(* CODESYS project xlh_gantry_example_1_00_02.project
   Author: 3S - Smart Software Solutions GmbH
   Version: 1.0.0.0
   Description: Receives some incoming messages and echoes them with CAN-ID +1
   Title: CAN Bus API Example
   Company: 3S - Smart Software Solutions GmbH

Project tree, tasks and I/O mapping:
  xLH_base : CODESYS Control for Raspberry Pi 64 SL, CODESYS, order no. 2302000009, version 4.20.0.0
    application app
      libraries: Standard, 3.5.22.0 (System); Util, 3.5.22.0 (System); VisuDialogs, * (System); Memory, * (3S - Smart Software Solutions GmbH); CmpBitmapPool, * (System); MemoryUtils, * (3S - Smart Software Solutions GmbH); CAA CiA 405, 4.3.0.0 (CODESYS)
      task CANOPEN_TASK (cyclic, interval 1 ms, priority 1) calls nothing
      task VISU_TASK (cyclic, interval 100 ms, priority 31) calls VisuElems.Visu_Prg
      task MAIN_TASK (cyclic, interval 4 ms, priority 2) calls io, MAIN_CALLER
      task SoftMotion_PlanningTask (cyclic, interval t#2ms, priority 15) calls nothing
      program MAIN_CALLER [ST]
      visualisation Visualization
      data type MOTION_CONTROL_BYTE
      MOTION_BASE/
        function block FB_XLH_MOTION_AXIS_SIMPLE_ES [ST]: mRead
        function block FB_PLC_OPEN_AXIS [ST]: plcOpen, executeToFalse
        function block FB_XLH_MOTION_AXIS_SIMPLE [ST]
        function block FB_XLH_MOTION_AXIS_BASE [ST]: mRead, mWrite
        function block FB_AXG_MOVE_ABSOLUTE [ST]
        function block FB_AXG_MOVE_RELATIVE [ST]
        function block FB_AXG_PICK_AND_PLACE [ST]: moveToOffset, setMagnet
        function block FB_KALMAN_FILTER [ST]: reset
        data type ST_PnpStep
      IO/
        function block FB_XLH_MOTION [ST]: read, write
        program io [ST]: read, write
        function block FB_XLH_GPIO [ST]: read, write
        function block FB_XLH_TERMINAL [ST]: read, write
        data type RGB
        data type UNION_BYTE_INT
        trace RT (task MAIN_TASK): io.terminal.bRtMagnet, io.terminal.bMagnet, MANUAL_MODE.iDummy
      program MC [ST]: write_io, read_io, axSmExecuteToFalse, axGexecuteToFalse, axInitPointers, axPowerOn, axStartHomingZA, axStopHoming, axCmdReset, axSetDefaultKinValues, axStartHomingXY, homing
      axis group AxisGroup: TRAFO.Kin_Gantry3, axes x_axis, y_axis, z_axis
      GCODE/
        text DEMO_GCODE
      CNC settings
      program MANUAL_MODE [ST]: TODO
      program CNC_MODE [ST]
      program APP_SQUARE_MODE [ST]
      MISC/
        TRACE/
          trace Trace_AxX (task MAIN_TASK): x_axis.fActPosition, x_axis.fSetPosition, x_axis.fSetAcceleration, x_axis.fActAcceleration, x_axis.fSetVelocity, x_axis.fActVelocity, io.motion.adiFrequency[1]
          trace Trace (task MAIN_TASK): MC.diPosition, MC.iSetSpeed, MC.iDebug2Pos, MC.iDebug1Mileage, MC.auiUltrasonic[1], MC.fbReadStatusLoopTime.udiValue, MC.iSpeed2, MC.iSpeed1, MC.iPitch
          trace Trace_AxZ (task MAIN_TASK): z_axis.fActPosition, z_axis.fSetPosition, z_axis.fSetAcceleration, z_axis.fActAcceleration, z_axis.fSetVelocity, z_axis.fActVelocity, io.motion.adiFrequency[3]
    CANbus : CANbus, CODESYS, version 4.3.0.0
        settings: Baudrate = 1000 kbit/s
      CANopen_Manager : CANopen_Manager, CODESYS, version 4.3.0.0
          settings: NMT Start All = TRUE; Polling of optional slaves = FALSE; ConfigVersion = 50659584
        xlh_motion : xlh_motion, xemax ag, order no. 0, version Revision=16#00000001, FileVersion=1.0
            settings: NODEIDSAVED = 1; SDO Timeout = 1000000; PDO_Autoconfig = FALSE; EXPERTSETTINGS = True; Sync-General Parameters.Sync-COBID = 16#00000080; Sync-General Parameters.Communication Cycle Period = 16#00000000 usec; PDO 16#1400.COBID = 16#00000201; Process by CANopenManager = TRUE; PDO 16#1401.COBID = 16#00000301; Process by CANopenManager = TRUE; PDO 16#1402.COBID = 16#00000401; Process by CANopenManager = TRUE; PDO 16#1403.COBID = 16#00000501; Process by CANopenManager = TRUE; PDO 16#1800.COBID = 16#00000181; Process by CANopenManager = TRUE; PDO 16#1801.COBID = 16#00000281; Process by CANopenManager = TRUE; PDO 16#1802.COBID = 16#00000381; Process by CANopenManager = TRUE; Control 1.Subindex = 16#01; Control 2.Subindex = 16#02; Control 3.Subindex = 16#03; Control 4.Subindex = 16#04; Outputs 0-7.Subindex = 16#01; Outputs 8-15.Subindex = 16#02; Magnet Duty Cycle.Subindex = 16#01; Freqeuncy 1.Subindex = 16#05; Freqeuncy 2.Subindex = 16#06; Freqeuncy 3.Subindex = 16#07; Freqeuncy 4.Subindex = 16#08; Servo 1.Subindex = 16#01; Servo 2.Subindex = 16#02; Servo 3.Subindex = 16#03; Servo 4.Subindex = 16#04; Servo 5.Subindex = 16#05; Servo 6.Subindex = 16#06; Servo 7.Subindex = 16#07; Servo 8.Subindex = 16#08; Position 1.Subindex = 16#01;
              Position 2.Subindex = 16#02; Position 3.Subindex = 16#03; Position 4.Subindex = 16#04; Inputs 0-7.Subindex = 16#01; Inputs 8-15.Subindex = 16#02; Inputs CLK.Subindex = 16#03; SDO List.Set COB-ID sync.Index = 16#1005; SDO List.Set COB-ID sync.Subindex = 16#00; SDO List.Set COB-ID sync.Value = 16#00000080; SDO List.Set COB-ID sync.Size = 32; SDO List.Set COB-ID sync.AbortIfError = FALSE; SDO List.Set COB-ID sync.JumpToLine = FALSE; SDO List.Set COB-ID sync.Line = 0; SDO List.Set communication cycle period.Index = 16#1006; SDO List.Set communication cycle period.Subindex = 16#00; SDO List.Set communication cycle period.Value = 16#00000000; SDO List.Set communication cycle period.Size = 32; SDO List.Set communication cycle period.AbortIfError = FALSE; SDO List.Set communication cycle period.JumpToLine = FALSE; SDO List.Set communication cycle period.Line = 0; SDO List.Set Guardtime.Index = 16#100C; SDO List.Set Guardtime.Subindex = 16#00; SDO List.Set Guardtime.Value = 16#000000C8; SDO List.Set Guardtime.Size = 16; SDO List.Set Guardtime.AbortIfError = FALSE; SDO List.Set Guardtime.JumpToLine = FALSE; SDO List.Set Guardtime.Line = 0; SDO List.Set Lifetime.Index = 16#100D; SDO List.Set Lifetime.Subindex = 16#00; SDO List.Set Lifetime.Value = 16#00000003; SDO List.Set Lifetime.Size = 8; SDO List.Set Lifetime.AbortIfError = FALSE; SDO List.Set Lifetime.JumpToLine = FALSE; SDO List.Set Lifetime.Line = 0; SDO List.Set Heartbeat Consumer.Index = 16#1016; SDO List.Set Heartbeat Consumer.Subindex = 16#01; SDO List.Set Heartbeat Consumer.Value = 0; SDO List.Set Heartbeat Consumer.Size = 32; SDO List.Set Heartbeat Consumer.AbortIfError = FALSE; SDO List.Set Heartbeat Consumer.JumpToLine = FALSE;
              SDO List.Set Heartbeat Consumer.Line = 0; SDO List.Disable PDO.Index = 16#1400; SDO List.Disable PDO.Subindex = 16#01; SDO List.Disable PDO.Value = 16#80000201; SDO List.Disable PDO.Size = 32; SDO List.Disable PDO.AbortIfError = FALSE; SDO List.Disable PDO.JumpToLine = FALSE; SDO List.Disable PDO.Line = 0; SDO List.Set transmission type.Index = 16#1400; SDO List.Set transmission type.Subindex = 16#02; SDO List.Set transmission type.Value = 16#FF; SDO List.Set transmission type.Size = 8; SDO List.Set transmission type.AbortIfError = FALSE; SDO List.Set transmission type.JumpToLine = FALSE; SDO List.Set transmission type.Line = 0; SDO List.Set and enable COB-ID.Index = 16#1400; SDO List.Set and enable COB-ID.Subindex = 16#01; SDO List.Set and enable COB-ID.Value = 16#00000201; SDO List.Set and enable COB-ID.Size = 32; SDO List.Set and enable COB-ID.AbortIfError = FALSE; SDO List.Set and enable COB-ID.JumpToLine = FALSE; SDO List.Set and enable COB-ID.Line = 0; SDO List.Disable PDO.Index = 16#1401; SDO List.Disable PDO.Subindex = 16#01; SDO List.Disable PDO.Value = 16#80000301; SDO List.Disable PDO.Size = 32; SDO List.Disable PDO.AbortIfError = FALSE; SDO List.Disable PDO.JumpToLine = FALSE; SDO List.Disable PDO.Line = 0; SDO List.Set transmission type.Index = 16#1401; SDO List.Set transmission type.Subindex = 16#02; SDO List.Set transmission type.Value = 16#FF; SDO List.Set transmission type.Size = 8; SDO List.Set transmission type.AbortIfError = FALSE; SDO List.Set transmission type.JumpToLine = FALSE; SDO List.Set transmission type.Line = 0; SDO List.Set and enable COB-ID.Index = 16#1401; SDO List.Set and enable COB-ID.Subindex = 16#01; SDO List.Set and enable COB-ID.Value = 16#00000301; SDO List.Set and enable COB-ID.Size = 32;
              SDO List.Set and enable COB-ID.AbortIfError = FALSE; SDO List.Set and enable COB-ID.JumpToLine = FALSE; SDO List.Set and enable COB-ID.Line = 0; SDO List.Disable PDO.Index = 16#1402; SDO List.Disable PDO.Subindex = 16#01; SDO List.Disable PDO.Value = 16#80000401; SDO List.Disable PDO.Size = 32; SDO List.Disable PDO.AbortIfError = FALSE; SDO List.Disable PDO.JumpToLine = FALSE; SDO List.Disable PDO.Line = 0; SDO List.Set transmission type.Index = 16#1402; SDO List.Set transmission type.Subindex = 16#02; SDO List.Set transmission type.Value = 16#FF; SDO List.Set transmission type.Size = 8; SDO List.Set transmission type.AbortIfError = FALSE; SDO List.Set transmission type.JumpToLine = FALSE; SDO List.Set transmission type.Line = 0; SDO List.Set and enable COB-ID.Index = 16#1402; SDO List.Set and enable COB-ID.Subindex = 16#01; SDO List.Set and enable COB-ID.Value = 16#00000401; SDO List.Set and enable COB-ID.Size = 32; SDO List.Set and enable COB-ID.AbortIfError = FALSE; SDO List.Set and enable COB-ID.JumpToLine = FALSE; SDO List.Set and enable COB-ID.Line = 0; SDO List.Disable PDO.Index = 16#1403; SDO List.Disable PDO.Subindex = 16#01; SDO List.Disable PDO.Value = 16#80000501; SDO List.Disable PDO.Size = 32; SDO List.Disable PDO.AbortIfError = FALSE; SDO List.Disable PDO.JumpToLine = FALSE; SDO List.Disable PDO.Line = 0; SDO List.Set transmission type.Index = 16#1403; SDO List.Set transmission type.Subindex = 16#02; SDO List.Set transmission type.Value = 16#FF; SDO List.Set transmission type.Size = 8; SDO List.Set transmission type.AbortIfError = FALSE; SDO List.Set transmission type.JumpToLine = FALSE; SDO List.Set transmission type.Line = 0; SDO List.Set and enable COB-ID.Index = 16#1403; SDO List.Set and enable COB-ID.Subindex = 16#01;
              SDO List.Set and enable COB-ID.Value = 16#00000501; SDO List.Set and enable COB-ID.Size = 32; SDO List.Set and enable COB-ID.AbortIfError = FALSE; SDO List.Set and enable COB-ID.JumpToLine = FALSE; SDO List.Set and enable COB-ID.Line = 0; SDO List.Disable PDO.Index = 16#1800; SDO List.Disable PDO.Subindex = 16#01; SDO List.Disable PDO.Value = 16#80000181; SDO List.Disable PDO.Size = 32; SDO List.Disable PDO.AbortIfError = FALSE; SDO List.Disable PDO.JumpToLine = FALSE; SDO List.Disable PDO.Line = 0; SDO List.Set transmission type.Index = 16#1800; SDO List.Set transmission type.Subindex = 16#02; SDO List.Set transmission type.Value = 16#FF; SDO List.Set transmission type.Size = 8; SDO List.Set transmission type.AbortIfError = FALSE; SDO List.Set transmission type.JumpToLine = FALSE; SDO List.Set transmission type.Line = 0; SDO List.Set inhibit time.Index = 16#1800; SDO List.Set inhibit time.Subindex = 16#03; SDO List.Set inhibit time.Value = 16#0000; SDO List.Set inhibit time.Size = 16; SDO List.Set inhibit time.AbortIfError = FALSE; SDO List.Set inhibit time.JumpToLine = FALSE; SDO List.Set inhibit time.Line = 0; SDO List.Set event time.Index = 16#1800; SDO List.Set event time.Subindex = 16#05; SDO List.Set event time.Value = 16#0000; SDO List.Set event time.Size = 16; SDO List.Set event time.AbortIfError = FALSE; SDO List.Set event time.JumpToLine = FALSE; SDO List.Set event time.Line = 0; SDO List.Set and enable COB-ID.Index = 16#1800; SDO List.Set and enable COB-ID.Subindex = 16#01; SDO List.Set and enable COB-ID.Value = 16#00000181; SDO List.Set and enable COB-ID.Size = 32; SDO List.Set and enable COB-ID.AbortIfError = FALSE; SDO List.Set and enable COB-ID.JumpToLine = FALSE; SDO List.Set and enable COB-ID.Line = 0;
              SDO List.Disable PDO.Index = 16#1801; SDO List.Disable PDO.Subindex = 16#01; SDO List.Disable PDO.Value = 16#80000281; SDO List.Disable PDO.Size = 32; SDO List.Disable PDO.AbortIfError = FALSE; SDO List.Disable PDO.JumpToLine = FALSE; SDO List.Disable PDO.Line = 0; SDO List.Set transmission type.Index = 16#1801; SDO List.Set transmission type.Subindex = 16#02; SDO List.Set transmission type.Value = 16#FF; SDO List.Set transmission type.Size = 8; SDO List.Set transmission type.AbortIfError = FALSE; SDO List.Set transmission type.JumpToLine = FALSE; SDO List.Set transmission type.Line = 0; SDO List.Set inhibit time.Index = 16#1801; SDO List.Set inhibit time.Subindex = 16#03; SDO List.Set inhibit time.Value = 16#0000; SDO List.Set inhibit time.Size = 16; SDO List.Set inhibit time.AbortIfError = FALSE; SDO List.Set inhibit time.JumpToLine = FALSE; SDO List.Set inhibit time.Line = 0; SDO List.Set event time.Index = 16#1801; SDO List.Set event time.Subindex = 16#05; SDO List.Set event time.Value = 16#0000; SDO List.Set event time.Size = 16; SDO List.Set event time.AbortIfError = FALSE; SDO List.Set event time.JumpToLine = FALSE; SDO List.Set event time.Line = 0; SDO List.Set and enable COB-ID.Index = 16#1801; SDO List.Set and enable COB-ID.Subindex = 16#01; SDO List.Set and enable COB-ID.Value = 16#00000281; SDO List.Set and enable COB-ID.Size = 32; SDO List.Set and enable COB-ID.AbortIfError = FALSE; SDO List.Set and enable COB-ID.JumpToLine = FALSE; SDO List.Set and enable COB-ID.Line = 0; SDO List.Disable PDO.Index = 16#1802; SDO List.Disable PDO.Subindex = 16#01; SDO List.Disable PDO.Value = 16#80000381; SDO List.Disable PDO.Size = 32; SDO List.Disable PDO.AbortIfError = FALSE;
              SDO List.Disable PDO.JumpToLine = FALSE; SDO List.Disable PDO.Line = 0; SDO List.Set transmission type.Index = 16#1802; SDO List.Set transmission type.Subindex = 16#02; SDO List.Set transmission type.Value = 16#FF; SDO List.Set transmission type.Size = 8; SDO List.Set transmission type.AbortIfError = FALSE; SDO List.Set transmission type.JumpToLine = FALSE; SDO List.Set transmission type.Line = 0; SDO List.Set inhibit time.Index = 16#1802; SDO List.Set inhibit time.Subindex = 16#03; SDO List.Set inhibit time.Value = 16#0000; SDO List.Set inhibit time.Size = 16; SDO List.Set inhibit time.AbortIfError = FALSE; SDO List.Set inhibit time.JumpToLine = FALSE; SDO List.Set inhibit time.Line = 0; SDO List.Set event time.Index = 16#1802; SDO List.Set event time.Subindex = 16#05; SDO List.Set event time.Value = 16#0000; SDO List.Set event time.Size = 16; SDO List.Set event time.AbortIfError = FALSE; SDO List.Set event time.JumpToLine = FALSE; SDO List.Set event time.Line = 0; SDO List.Set and enable COB-ID.Index = 16#1802; SDO List.Set and enable COB-ID.Subindex = 16#01; SDO List.Set and enable COB-ID.Value = 16#00000381; SDO List.Set and enable COB-ID.Size = 32; SDO List.Set and enable COB-ID.AbortIfError = FALSE; SDO List.Set and enable COB-ID.JumpToLine = FALSE; SDO List.Set and enable COB-ID.Line = 0; ConfigVersion = 50659584
            output app.io.motion.abyControl[1] : USINT  // Control 1
            output app.io.motion.abyControl[2] : USINT  // Control 2
            output app.io.motion.abyControl[3] : USINT  // Control 3
            output app.io.motion.abyControl[4] : USINT  // Control 4
            output app.io.motion.abyOutputs[1] : USINT  // Outputs 0-7
            output app.io.motion.abyOutputs[2] : USINT  // Outputs 8-15
            output app.io.motion.uiMagnetDutyCycle : UINT  // Magnet Duty Cycle
            output app.io.motion.adiFrequency[1] : DINT  // Freqeuncy 1
            output app.io.motion.adiFrequency[2] : DINT  // Freqeuncy 2
            output app.io.motion.adiFrequency[3] : DINT  // Freqeuncy 3
            output app.io.motion.adiFrequency[4] : DINT  // Freqeuncy 4
            output app.io.motion.ausServo[1] : USINT  // Servo 1
            output app.io.motion.ausServo[2] : USINT  // Servo 2
            output app.io.motion.ausServo[3] : USINT  // Servo 3
            output app.io.motion.ausServo[4] : USINT  // Servo 4
            output app.io.motion.ausServo[5] : USINT  // Servo 5
            output app.io.motion.ausServo[6] : USINT  // Servo 6
            output app.io.motion.ausServo[7] : USINT  // Servo 7
            output app.io.motion.ausServo[8] : USINT  // Servo 8
            input  app.io.motion.adiPosition[1] : DINT  // Position 1
            input  app.io.motion.adiPosition[2] : DINT  // Position 2
            input  app.io.motion.adiPosition[3] : DINT  // Position 3
            input  app.io.motion.adiPosition[4] : DINT  // Position 4
            input  app.io.motion.abyInputs[1] : USINT  // Inputs 0-7
            input  app.io.motion.bAxXsw : BOOL  // Inputs 0-7.Bit0
            input  app.io.motion.bAxYsw : BOOL  // Inputs 0-7.Bit1
            input  app.io.motion.bAxZsw : BOOL  // Inputs 0-7.Bit2
            input  app.io.motion._bSensorHw : BOOL  // Inputs 0-7.Bit3
            input  app.io.motion._bSensorConveyorFrontHw : BOOL  // Inputs 0-7.Bit4
            input  app.io.motion._bSensorConveyorBackHw : BOOL  // Inputs 0-7.Bit5
            input  app.io.motion.abyInputs[2] : USINT  // Inputs 8-15
            input  app.io.motion.abyInputs[3] : USINT  // Inputs CLK
        xlh_terminal : xlh_terminal, xemax ag, order no. 0, version Revision=16#00000001, FileVersion=1.0
            settings: NODEIDSAVED = 2; SDO Timeout = 1000000; PDO_Autoconfig = FALSE; EXPERTSETTINGS = FALSE; Nodeguarding.Guard Time = 1000 ms; PDO 16#1400.COBID = 16#00000202; Process by CANopenManager = TRUE; PDO 16#1401.COBID = 16#00000302; Process by CANopenManager = TRUE; PDO 16#1402.COBID = 16#00000402; Process by CANopenManager = TRUE; PDO 16#1403.COBID = 16#00000502; Process by CANopenManager = TRUE; PDO 16#1800.COBID = 16#00000182; Process by CANopenManager = TRUE; PDO 16#1801.COBID = 16#00000282; Process by CANopenManager = TRUE; PDO 16#1802.COBID = 16#00000382; Process by CANopenManager = TRUE; PDO 16#1803.COBID = 16#00000482; Process by CANopenManager = TRUE; Data out 1 Byte 0.Subindex = 16#01; Data out 1 Byte 1.Subindex = 16#02; Data out 1 Byte 2.Subindex = 16#03; Data out 1 Byte 3.Subindex = 16#04; Data out 1 Byte 4.Subindex = 16#05; Data out 1 Byte 5.Subindex = 16#06; Data out 1 Byte 6.Subindex = 16#07; Data out 1 Byte 7.Subindex = 16#08; Data out 2 Byte 0.Subindex = 16#01; Data out 2 Byte 1.Subindex = 16#02; Data out 2 Byte 2.Subindex = 16#03; Data out 2 Byte 3.Subindex = 16#04; Data out 2 Byte 4.Subindex = 16#05; Data out 2 Byte 5.Subindex = 16#06; Data out 2 Byte 6.Subindex = 16#07; Data out 2 Byte 7.Subindex = 16#08; Data out 3 Byte 0.Subindex = 16#01; Data out 3 Byte 1.Subindex = 16#02; Data out 3 Byte 2.Subindex = 16#03;
              Data out 3 Byte 3.Subindex = 16#04; Data out 3 Byte 4.Subindex = 16#05; Data out 3 Byte 5.Subindex = 16#06; Data out 3 Byte 6.Subindex = 16#07; Data out 3 Byte 7.Subindex = 16#08; Data out 4 Byte 0.Subindex = 16#01; Data out 4 Byte 1.Subindex = 16#02; Data out 4 Byte 2.Subindex = 16#03; Data out 4 Byte 3.Subindex = 16#04; Data out 4 Byte 4.Subindex = 16#05; Data out 4 Byte 5.Subindex = 16#06; Data out 4 Byte 6.Subindex = 16#07; Data out 4 Byte 7.Subindex = 16#08; Data in 1 Byte 0.Subindex = 16#01; Data in 1 Byte 1.Subindex = 16#02; Data in 1 Byte 2.Subindex = 16#03; Data in 1 Byte 3.Subindex = 16#04; Data in 1 Byte 4.Subindex = 16#05; Data in 1 Byte 5.Subindex = 16#06; Data in 1 Byte 6.Subindex = 16#07; Data in 1 Byte 7.Subindex = 16#08; Data in 2 Byte 0.Subindex = 16#01; Data in 2 Byte 1.Subindex = 16#02; Data in 2 Byte 2.Subindex = 16#03; Data in 2 Byte 3.Subindex = 16#04; Data in 2 Byte 4.Subindex = 16#05; Data in 2 Byte 5.Subindex = 16#06; Data in 2 Byte 6.Subindex = 16#07; Data in 2 Byte 7.Subindex = 16#08; Data in 3 Byte 0.Subindex = 16#01; Data in 3 Byte 1.Subindex = 16#02; Data in 3 Byte 2.Subindex = 16#03; Data in 3 Byte 3.Subindex = 16#04; Data in 3 Byte 4.Subindex = 16#05; Data in 3 Byte 5.Subindex = 16#06; Data in 3 Byte 6.Subindex = 16#07; Data in 3 Byte 7.Subindex = 16#08; Data in 4 Byte 0.Subindex = 16#01; Data in 4 Byte 1.Subindex = 16#02; Data in 4 Byte 2.Subindex = 16#03;
              Data in 4 Byte 3.Subindex = 16#04; Data in 4 Byte 4.Subindex = 16#05; Data in 4 Byte 5.Subindex = 16#06; Data in 4 Byte 6.Subindex = 16#07; Data in 4 Byte 7.Subindex = 16#08; SDO List.Set COB-ID sync.Index = 16#1005; SDO List.Set COB-ID sync.Subindex = 16#00; SDO List.Set COB-ID sync.Value = 16#00000080; SDO List.Set COB-ID sync.Size = 32; SDO List.Set COB-ID sync.AbortIfError = FALSE; SDO List.Set COB-ID sync.JumpToLine = FALSE; SDO List.Set COB-ID sync.Line = 0; SDO List.Set communication cycle period.Index = 16#1006; SDO List.Set communication cycle period.Subindex = 16#00; SDO List.Set communication cycle period.Value = 16#00000000; SDO List.Set communication cycle period.Size = 32; SDO List.Set communication cycle period.AbortIfError = FALSE; SDO List.Set communication cycle period.JumpToLine = FALSE; SDO List.Set communication cycle period.Line = 0; SDO List.Set Guardtime.Index = 16#100C; SDO List.Set Guardtime.Subindex = 16#00; SDO List.Set Guardtime.Value = 16#000003E8; SDO List.Set Guardtime.Size = 16; SDO List.Set Guardtime.AbortIfError = FALSE; SDO List.Set Guardtime.JumpToLine = FALSE; SDO List.Set Guardtime.Line = 0; SDO List.Set Lifetime.Index = 16#100D; SDO List.Set Lifetime.Subindex = 16#00; SDO List.Set Lifetime.Value = 16#00000003; SDO List.Set Lifetime.Size = 8; SDO List.Set Lifetime.AbortIfError = FALSE; SDO List.Set Lifetime.JumpToLine = FALSE; SDO List.Set Lifetime.Line = 0; SDO List.Set Heartbeat Consumer.Index = 16#1016; SDO List.Set Heartbeat Consumer.Subindex = 16#01; SDO List.Set Heartbeat Consumer.Value = 0; SDO List.Set Heartbeat Consumer.Size = 32; SDO List.Set Heartbeat Consumer.AbortIfError = FALSE; SDO List.Set Heartbeat Consumer.JumpToLine = FALSE; SDO List.Set Heartbeat Consumer.Line = 0;
              SDO List.Disable PDO.Index = 16#1400; SDO List.Disable PDO.Subindex = 16#01; SDO List.Disable PDO.Value = 16#80000202; SDO List.Disable PDO.Size = 32; SDO List.Disable PDO.AbortIfError = FALSE; SDO List.Disable PDO.JumpToLine = FALSE; SDO List.Disable PDO.Line = 0; SDO List.Set transmission type.Index = 16#1400; SDO List.Set transmission type.Subindex = 16#02; SDO List.Set transmission type.Value = 16#FF; SDO List.Set transmission type.Size = 8; SDO List.Set transmission type.AbortIfError = FALSE; SDO List.Set transmission type.JumpToLine = FALSE; SDO List.Set transmission type.Line = 0; SDO List.Set and enable COB-ID.Index = 16#1400; SDO List.Set and enable COB-ID.Subindex = 16#01; SDO List.Set and enable COB-ID.Value = 16#00000202; SDO List.Set and enable COB-ID.Size = 32; SDO List.Set and enable COB-ID.AbortIfError = FALSE; SDO List.Set and enable COB-ID.JumpToLine = FALSE; SDO List.Set and enable COB-ID.Line = 0; SDO List.Disable PDO.Index = 16#1401; SDO List.Disable PDO.Subindex = 16#01; SDO List.Disable PDO.Value = 16#80000302; SDO List.Disable PDO.Size = 32; SDO List.Disable PDO.AbortIfError = FALSE; SDO List.Disable PDO.JumpToLine = FALSE; SDO List.Disable PDO.Line = 0; SDO List.Set transmission type.Index = 16#1401; SDO List.Set transmission type.Subindex = 16#02; SDO List.Set transmission type.Value = 16#FF; SDO List.Set transmission type.Size = 8; SDO List.Set transmission type.AbortIfError = FALSE; SDO List.Set transmission type.JumpToLine = FALSE; SDO List.Set transmission type.Line = 0; SDO List.Set and enable COB-ID.Index = 16#1401; SDO List.Set and enable COB-ID.Subindex = 16#01; SDO List.Set and enable COB-ID.Value = 16#00000302; SDO List.Set and enable COB-ID.Size = 32; SDO List.Set and enable COB-ID.AbortIfError = FALSE;
              SDO List.Set and enable COB-ID.JumpToLine = FALSE; SDO List.Set and enable COB-ID.Line = 0; SDO List.Disable PDO.Index = 16#1402; SDO List.Disable PDO.Subindex = 16#01; SDO List.Disable PDO.Value = 16#80000402; SDO List.Disable PDO.Size = 32; SDO List.Disable PDO.AbortIfError = FALSE; SDO List.Disable PDO.JumpToLine = FALSE; SDO List.Disable PDO.Line = 0; SDO List.Set transmission type.Index = 16#1402; SDO List.Set transmission type.Subindex = 16#02; SDO List.Set transmission type.Value = 16#FF; SDO List.Set transmission type.Size = 8; SDO List.Set transmission type.AbortIfError = FALSE; SDO List.Set transmission type.JumpToLine = FALSE; SDO List.Set transmission type.Line = 0; SDO List.Set and enable COB-ID.Index = 16#1402; SDO List.Set and enable COB-ID.Subindex = 16#01; SDO List.Set and enable COB-ID.Value = 16#00000402; SDO List.Set and enable COB-ID.Size = 32; SDO List.Set and enable COB-ID.AbortIfError = FALSE; SDO List.Set and enable COB-ID.JumpToLine = FALSE; SDO List.Set and enable COB-ID.Line = 0; SDO List.Disable PDO.Index = 16#1403; SDO List.Disable PDO.Subindex = 16#01; SDO List.Disable PDO.Value = 16#80000502; SDO List.Disable PDO.Size = 32; SDO List.Disable PDO.AbortIfError = FALSE; SDO List.Disable PDO.JumpToLine = FALSE; SDO List.Disable PDO.Line = 0; SDO List.Set transmission type.Index = 16#1403; SDO List.Set transmission type.Subindex = 16#02; SDO List.Set transmission type.Value = 16#FF; SDO List.Set transmission type.Size = 8; SDO List.Set transmission type.AbortIfError = FALSE; SDO List.Set transmission type.JumpToLine = FALSE; SDO List.Set transmission type.Line = 0; SDO List.Set and enable COB-ID.Index = 16#1403; SDO List.Set and enable COB-ID.Subindex = 16#01; SDO List.Set and enable COB-ID.Value = 16#00000502;
              SDO List.Set and enable COB-ID.Size = 32; SDO List.Set and enable COB-ID.AbortIfError = FALSE; SDO List.Set and enable COB-ID.JumpToLine = FALSE; SDO List.Set and enable COB-ID.Line = 0; SDO List.Disable PDO.Index = 16#1800; SDO List.Disable PDO.Subindex = 16#01; SDO List.Disable PDO.Value = 16#80000182; SDO List.Disable PDO.Size = 32; SDO List.Disable PDO.AbortIfError = FALSE; SDO List.Disable PDO.JumpToLine = FALSE; SDO List.Disable PDO.Line = 0; SDO List.Set transmission type.Index = 16#1800; SDO List.Set transmission type.Subindex = 16#02; SDO List.Set transmission type.Value = 16#FF; SDO List.Set transmission type.Size = 8; SDO List.Set transmission type.AbortIfError = FALSE; SDO List.Set transmission type.JumpToLine = FALSE; SDO List.Set transmission type.Line = 0; SDO List.Set inhibit time.Index = 16#1800; SDO List.Set inhibit time.Subindex = 16#03; SDO List.Set inhibit time.Value = 16#0000; SDO List.Set inhibit time.Size = 16; SDO List.Set inhibit time.AbortIfError = FALSE; SDO List.Set inhibit time.JumpToLine = FALSE; SDO List.Set inhibit time.Line = 0; SDO List.Set event time.Index = 16#1800; SDO List.Set event time.Subindex = 16#05; SDO List.Set event time.Value = 16#0000; SDO List.Set event time.Size = 16; SDO List.Set event time.AbortIfError = FALSE; SDO List.Set event time.JumpToLine = FALSE; SDO List.Set event time.Line = 0; SDO List.Set and enable COB-ID.Index = 16#1800; SDO List.Set and enable COB-ID.Subindex = 16#01; SDO List.Set and enable COB-ID.Value = 16#00000182; SDO List.Set and enable COB-ID.Size = 32; SDO List.Set and enable COB-ID.AbortIfError = FALSE; SDO List.Set and enable COB-ID.JumpToLine = FALSE; SDO List.Set and enable COB-ID.Line = 0; SDO List.Disable PDO.Index = 16#1801;
              SDO List.Disable PDO.Subindex = 16#01; SDO List.Disable PDO.Value = 16#80000282; SDO List.Disable PDO.Size = 32; SDO List.Disable PDO.AbortIfError = FALSE; SDO List.Disable PDO.JumpToLine = FALSE; SDO List.Disable PDO.Line = 0; SDO List.Set transmission type.Index = 16#1801; SDO List.Set transmission type.Subindex = 16#02; SDO List.Set transmission type.Value = 16#FF; SDO List.Set transmission type.Size = 8; SDO List.Set transmission type.AbortIfError = FALSE; SDO List.Set transmission type.JumpToLine = FALSE; SDO List.Set transmission type.Line = 0; SDO List.Set inhibit time.Index = 16#1801; SDO List.Set inhibit time.Subindex = 16#03; SDO List.Set inhibit time.Value = 16#0000; SDO List.Set inhibit time.Size = 16; SDO List.Set inhibit time.AbortIfError = FALSE; SDO List.Set inhibit time.JumpToLine = FALSE; SDO List.Set inhibit time.Line = 0; SDO List.Set event time.Index = 16#1801; SDO List.Set event time.Subindex = 16#05; SDO List.Set event time.Value = 16#0000; SDO List.Set event time.Size = 16; SDO List.Set event time.AbortIfError = FALSE; SDO List.Set event time.JumpToLine = FALSE; SDO List.Set event time.Line = 0; SDO List.Set and enable COB-ID.Index = 16#1801; SDO List.Set and enable COB-ID.Subindex = 16#01; SDO List.Set and enable COB-ID.Value = 16#00000282; SDO List.Set and enable COB-ID.Size = 32; SDO List.Set and enable COB-ID.AbortIfError = FALSE; SDO List.Set and enable COB-ID.JumpToLine = FALSE; SDO List.Set and enable COB-ID.Line = 0; SDO List.Disable PDO.Index = 16#1802; SDO List.Disable PDO.Subindex = 16#01; SDO List.Disable PDO.Value = 16#80000382; SDO List.Disable PDO.Size = 32; SDO List.Disable PDO.AbortIfError = FALSE; SDO List.Disable PDO.JumpToLine = FALSE;
              SDO List.Disable PDO.Line = 0; SDO List.Set transmission type.Index = 16#1802; SDO List.Set transmission type.Subindex = 16#02; SDO List.Set transmission type.Value = 16#FF; SDO List.Set transmission type.Size = 8; SDO List.Set transmission type.AbortIfError = FALSE; SDO List.Set transmission type.JumpToLine = FALSE; SDO List.Set transmission type.Line = 0; SDO List.Set inhibit time.Index = 16#1802; SDO List.Set inhibit time.Subindex = 16#03; SDO List.Set inhibit time.Value = 16#0000; SDO List.Set inhibit time.Size = 16; SDO List.Set inhibit time.AbortIfError = FALSE; SDO List.Set inhibit time.JumpToLine = FALSE; SDO List.Set inhibit time.Line = 0; SDO List.Set event time.Index = 16#1802; SDO List.Set event time.Subindex = 16#05; SDO List.Set event time.Value = 16#0000; SDO List.Set event time.Size = 16; SDO List.Set event time.AbortIfError = FALSE; SDO List.Set event time.JumpToLine = FALSE; SDO List.Set event time.Line = 0; SDO List.Set and enable COB-ID.Index = 16#1802; SDO List.Set and enable COB-ID.Subindex = 16#01; SDO List.Set and enable COB-ID.Value = 16#00000382; SDO List.Set and enable COB-ID.Size = 32; SDO List.Set and enable COB-ID.AbortIfError = FALSE; SDO List.Set and enable COB-ID.JumpToLine = FALSE; SDO List.Set and enable COB-ID.Line = 0; SDO List.Disable PDO.Index = 16#1803; SDO List.Disable PDO.Subindex = 16#01; SDO List.Disable PDO.Value = 16#80000482; SDO List.Disable PDO.Size = 32; SDO List.Disable PDO.AbortIfError = FALSE; SDO List.Disable PDO.JumpToLine = FALSE; SDO List.Disable PDO.Line = 0; SDO List.Set transmission type.Index = 16#1803; SDO List.Set transmission type.Subindex = 16#02; SDO List.Set transmission type.Value = 16#FF; SDO List.Set transmission type.Size = 8;
              SDO List.Set transmission type.AbortIfError = FALSE; SDO List.Set transmission type.JumpToLine = FALSE; SDO List.Set transmission type.Line = 0; SDO List.Set inhibit time.Index = 16#1803; SDO List.Set inhibit time.Subindex = 16#03; SDO List.Set inhibit time.Value = 16#0000; SDO List.Set inhibit time.Size = 16; SDO List.Set inhibit time.AbortIfError = FALSE; SDO List.Set inhibit time.JumpToLine = FALSE; SDO List.Set inhibit time.Line = 0; SDO List.Set event time.Index = 16#1803; SDO List.Set event time.Subindex = 16#05; SDO List.Set event time.Value = 16#0000; SDO List.Set event time.Size = 16; SDO List.Set event time.AbortIfError = FALSE; SDO List.Set event time.JumpToLine = FALSE; SDO List.Set event time.Line = 0; SDO List.Set and enable COB-ID.Index = 16#1803; SDO List.Set and enable COB-ID.Subindex = 16#01; SDO List.Set and enable COB-ID.Value = 16#00000482; SDO List.Set and enable COB-ID.Size = 32; SDO List.Set and enable COB-ID.AbortIfError = FALSE; SDO List.Set and enable COB-ID.JumpToLine = FALSE; SDO List.Set and enable COB-ID.Line = 0; ConfigVersion = 50659584
            output app.io.terminal.abyOutData1[0] : USINT  // Data out 1 Byte 0
            output app.io.terminal.abyOutData1[1] : USINT  // Data out 1 Byte 1
            output app.io.terminal.abyOutData1[2] : USINT  // Data out 1 Byte 2
            output app.io.terminal.abyOutData1[3] : USINT  // Data out 1 Byte 3
            output app.io.terminal.abyOutData1[4] : USINT  // Data out 1 Byte 4
            output app.io.terminal.abyOutData1[5] : USINT  // Data out 1 Byte 5
            output app.io.terminal.abyOutData1[6] : USINT  // Data out 1 Byte 6
            output app.io.terminal.abyOutData1[7] : USINT  // Data out 1 Byte 7
            output app.io.terminal.abyOutData2[0] : USINT  // Data out 2 Byte 0
            output app.io.terminal.abyOutData2[1] : USINT  // Data out 2 Byte 1
            output app.io.terminal.abyOutData2[2] : USINT  // Data out 2 Byte 2
            output app.io.terminal.abyOutData2[3] : USINT  // Data out 2 Byte 3
            output app.io.terminal.abyOutData2[4] : USINT  // Data out 2 Byte 4
            output app.io.terminal.abyOutData2[5] : USINT  // Data out 2 Byte 5
            output app.io.terminal.abyOutData2[6] : USINT  // Data out 2 Byte 6
            output app.io.terminal.abyOutData2[7] : USINT  // Data out 2 Byte 7
            output app.io.terminal.abyOutData3[0] : USINT  // Data out 3 Byte 0
            output app.io.terminal.abyOutData3[1] : USINT  // Data out 3 Byte 1
            output app.io.terminal.abyOutData3[2] : USINT  // Data out 3 Byte 2
            output app.io.terminal.abyOutData3[3] : USINT  // Data out 3 Byte 3
            output app.io.terminal.abyOutData3[4] : USINT  // Data out 3 Byte 4
            output app.io.terminal.abyOutData3[5] : USINT  // Data out 3 Byte 5
            output app.io.terminal.abyOutData3[6] : USINT  // Data out 3 Byte 6
            output app.io.terminal.abyOutData3[7] : USINT  // Data out 3 Byte 7
            output app.io.terminal.abyOutData4[0] : USINT  // Data out 4 Byte 0
            output app.io.terminal.abyOutData4[1] : USINT  // Data out 4 Byte 1
            output app.io.terminal.abyOutData4[2] : USINT  // Data out 4 Byte 2
            output app.io.terminal.abyOutData4[3] : USINT  // Data out 4 Byte 3
            output app.io.terminal.abyOutData4[4] : USINT  // Data out 4 Byte 4
            output app.io.terminal.abyOutData4[5] : USINT  // Data out 4 Byte 5
            output app.io.terminal.abyOutData4[6] : USINT  // Data out 4 Byte 6
            output app.io.terminal.abyOutData4[7] : USINT  // Data out 4 Byte 7
            input  app.io.terminal.abyInData1[0] : USINT  // Data in 1 Byte 0
            input  app.io.terminal.abyInData1[1] : USINT  // Data in 1 Byte 1
            input  app.io.terminal.abyInData1[2] : USINT  // Data in 1 Byte 2
            input  app.io.terminal.abyInData1[3] : USINT  // Data in 1 Byte 3
            input  app.io.terminal.abyInData1[4] : USINT  // Data in 1 Byte 4
            input  app.io.terminal.abyInData1[5] : USINT  // Data in 1 Byte 5
            input  app.io.terminal.abyInData1[6] : USINT  // Data in 1 Byte 6
            input  app.io.terminal.abyInData1[7] : USINT  // Data in 1 Byte 7
            input  app.io.terminal.abyInData2[0] : USINT  // Data in 2 Byte 0
            input  app.io.terminal.abyInData2[1] : USINT  // Data in 2 Byte 1
            input  app.io.terminal.abyInData2[2] : USINT  // Data in 2 Byte 2
            input  app.io.terminal.abyInData2[3] : USINT  // Data in 2 Byte 3
            input  app.io.terminal.abyInData2[4] : USINT  // Data in 2 Byte 4
            input  app.io.terminal.abyInData2[5] : USINT  // Data in 2 Byte 5
            input  app.io.terminal.abyInData2[6] : USINT  // Data in 2 Byte 6
            input  app.io.terminal.abyInData2[7] : USINT  // Data in 2 Byte 7
            input  app.io.terminal.abyInData3[0] : USINT  // Data in 3 Byte 0
            input  app.io.terminal.abyInData3[1] : USINT  // Data in 3 Byte 1
            input  app.io.terminal.abyInData3[2] : USINT  // Data in 3 Byte 2
            input  app.io.terminal.abyInData3[3] : USINT  // Data in 3 Byte 3
            input  app.io.terminal.abyInData3[4] : USINT  // Data in 3 Byte 4
            input  app.io.terminal.abyInData3[5] : USINT  // Data in 3 Byte 5
            input  app.io.terminal.abyInData3[6] : USINT  // Data in 3 Byte 6
            input  app.io.terminal.abyInData3[7] : USINT  // Data in 3 Byte 7
            input  app.io.terminal.abyInData4[0] : USINT  // Data in 4 Byte 0
            input  app.io.terminal.abyInData4[1] : USINT  // Data in 4 Byte 1
            input  app.io.terminal.abyInData4[2] : USINT  // Data in 4 Byte 2
            input  app.io.terminal.abyInData4[3] : USINT  // Data in 4 Byte 3
            input  app.io.terminal.abyInData4[4] : USINT  // Data in 4 Byte 4
            input  app.io.terminal.abyInData4[5] : USINT  // Data in 4 Byte 5
            input  app.io.terminal.abyInData4[6] : USINT  // Data in 4 Byte 6
            input  app.io.terminal.abyInData4[7] : USINT  // Data in 4 Byte 7
    Camera device
      <Leer>
    GPIOs_A_B : GPIOs B+/Pi2, CODESYS, version 4.20.0.0
        input  app.io.gpio.bSw1 : BOOL  // digital inputs (GPIO0..GPIO31).Bit4
        input  app.io.gpio.bSw2 : BOOL  // digital inputs (GPIO0..GPIO31).Bit5
        input  app.io.gpio.bSw3 : BOOL  // digital inputs (GPIO0..GPIO31).Bit6
        input  app.io.gpio.bSw4 : BOOL  // digital inputs (GPIO0..GPIO31).Bit12
        input  app.io.gpio.bSw5 : BOOL  // digital inputs (GPIO0..GPIO31).Bit13
        input  app.io.gpio.bSw6 : BOOL  // digital inputs (GPIO0..GPIO31).Bit16
        input  app.io.gpio.bSw7 : BOOL  // digital inputs (GPIO0..GPIO31).Bit17
        input  app.io.gpio.bSw8 : BOOL  // digital inputs (GPIO0..GPIO31).Bit19
        output app.io.gpio.bLed1 : BOOL  // digital outputs (GPIO0..GPIO31).Bit20
        output app.io.gpio.bLed2 : BOOL  // digital outputs (GPIO0..GPIO31).Bit21
        output app.io.gpio.bLed3 : BOOL  // digital outputs (GPIO0..GPIO31).Bit22
        output app.io.gpio.bLed4 : BOOL  // digital outputs (GPIO0..GPIO31).Bit23
        output app.io.gpio.bLed5 : BOOL  // digital outputs (GPIO0..GPIO31).Bit24
        output app.io.gpio.bLed6 : BOOL  // digital outputs (GPIO0..GPIO31).Bit26
        output app.io.gpio.bLed7 : BOOL  // digital outputs (GPIO0..GPIO31).Bit27
        unmapped channels: digital inputs (GPIO0..GPIO31), digital outputs (GPIO0..GPIO31)
    I²C
    SoftMotion General Axis Pool
      x_axis : SM_Drive_PosControl, CODESYS, order no. 1805, version 4.18.0.0
          settings: wDriveID = 0; dwRatioTechUnitsDenom = 101846; iRatioTechUnitsNum = 125; eRampType = 0; fSWMaxVelocity = 50; fSWMaxAcceleration = 100; fSWMaxDeceleration = 100; fSWMaxJerk = 1000; fSWLimitNegative = -1000; ScalingIncs = 814768; ScalingUnits = 1000; IsLinearMotor = TRUE; MaximumOutputVelocityInt = 40738; MinimumOutputVelocityInt = -40738; Kp = 0.005; MaxFollowingError = 1; PartVelocityPilotControl = 1; DeadTime = 1
      z_axis : SM_Drive_PosControl, CODESYS, order no. 1805, version 4.18.0.0
          settings: wDriveID = 2; dwRatioTechUnitsDenom = 101846; iRatioTechUnitsNum = -125; eRampType = 0; fSWMaxVelocity = 50; fSWMaxAcceleration = 100; fSWMaxDeceleration = 100; fSWMaxJerk = 1000; fSWLimitNegative = -1000; ScalingIncs = 814768; ScalingUnits = 1000; InvertDirection = TRUE; IsLinearMotor = TRUE; MaximumOutputVelocityInt = 40738; MinimumOutputVelocityInt = -40738; Kp = 0.005; MaxFollowingError = 1; DeadTime = 1
      y_axis : SM_Drive_PosControl, CODESYS, order no. 1805, version 4.18.0.0
          settings: dwRatioTechUnitsDenom = 101846; iRatioTechUnitsNum = -125; eRampType = 0; fSWMaxVelocity = 50; fSWMaxAcceleration = 100; fSWMaxDeceleration = 100; fSWMaxJerk = 1000; fSWLimitNegative = -1000; ScalingIncs = 814768; ScalingUnits = 1000; InvertDirection = TRUE; IsLinearMotor = TRUE; MaximumOutputVelocityInt = 40738; MinimumOutputVelocityInt = -40738; Kp = 0.005; MaxFollowingError = 1; PartVelocityPilotControl = 1; DeadTime = 1
      c_axis : SM_Drive_PosControl, CODESYS, order no. 1805, version 4.18.0.0
          settings: wDriveID = 3; dwRatioTechUnitsDenom = 530; iRatioTechUnitsNum = -1; eRampType = 0; fSWMaxVelocity = 50; fSWMaxAcceleration = 100; fSWMaxDeceleration = 100; fSWMaxJerk = 1000; fSWLimitNegative = -1000.0; ScalingIncs = 530000; ScalingUnits = 1000; InvertDirection = TRUE; IsLinearMotor = TRUE; MaximumOutputVelocityInt = 26000; MinimumOutputVelocityInt = -26000; Kp = 0.005; MaxFollowingError = 1; DeadTime = 1
    Onewire
    SPI
  libraries: VisuSymbols, 4.5.0.0 (System); DepictorBase, 1.2.0.0 (CODESYS)
  text list GlobalTextList
  5ce3da45-db07-42e7-a21c-a00fff4ed8f6|C:\Users\phe\Downloads\Musterloesung_FUP.PNG
*)

// xLH_base/app/MOTION_CONTROL_BYTE
TYPE MOTION_CONTROL_BYTE :
STRUCT
	bEnable: BOOL;
	bDir: BOOL;
	bReset: BOOL;
	bInverted: BOOL;
	bInMotion: BOOL;
	bMoveWithoutPulse: BOOL;
END_STRUCT
END_TYPE

// xLH_base/app/MOTION_BASE/ST_PnpStep
// =====================================================================
// ST_PnpStep
// Data structure for a single pick-and-place step.
// Contains the pick coordinates (fPickX/fPickY) and the place
// coordinates (fPlaceX/fPlaceY) in the XY plane. Used in the constant
// arrays PNP_STEPS and PNP_GRID of FB_PNP_SQUARE.
// =====================================================================
TYPE ST_PnpStep :
STRUCT
	fPickX  : LREAL;
	fPickY  : LREAL;
	fPlaceX : LREAL;
	fPlaceY : LREAL;
END_STRUCT
END_TYPE

// xLH_base/app/IO/RGB
{attribute 'qualified_only'}
{attribute 'strict'}
TYPE RGB :
(
	OFF := 0,
	RED := 1,
	GREEN := 2,
	BLUE := 3
);
END_TYPE

// xLH_base/app/IO/UNION_BYTE_INT
TYPE UNION_BYTE_INT :
UNION
	uiInt: UINT;;
	iInt: INT;
	abyStream: ARRAY[0..1] OF BYTE;	
END_UNION
END_TYPE

// xLH_base/app/IO/io
PROGRAM io 
VAR_INPUT
	gpio: FB_XLH_GPIO;	
	terminal: FB_XLH_TERMINAL;
	motion: FB_XLH_MOTION;
	bMagnet: BOOL;

	fbXlhMotionAxisX: FB_XLH_MOTION_AXIS_SIMPLE_ES;
	fbXlhMotionAxisY: FB_XLH_MOTION_AXIS_SIMPLE_ES;
	fbXlhMotionAxisZ: FB_XLH_MOTION_AXIS_SIMPLE_ES;
	fbXlhMotionAxisC: FB_XLH_MOTION_AXIS_SIMPLE;
END_VAR
VAR
	bStartup: BOOL := TRUE;
	i: INT;
END_VAR
VAR CONSTANT
	uiMAGNET_ON  : UINT := 4095;
	uiMAGNET_OFF : UINT := 0;
END_VAR

IF bStartup THEN
	bStartup := FALSE;

	io.motion.ausServo[1] := 128;

	fbXlhMotionAxisX.fbAxisPlcOpen REF= MC.axX;
	fbXlhMotionAxisX.pAxis         := ADR(x_axis);
	fbXlhMotionAxisX.pbEs          := ADR(io.motion.bAxXsw);

	fbXlhMotionAxisY.fbAxisPlcOpen REF= MC.axY;
	fbXlhMotionAxisY.pAxis         := ADR(y_axis);
	fbXlhMotionAxisY.pbEs          := ADR(io.motion.bAxYsw);

	fbXlhMotionAxisZ.fbAxisPlcOpen REF= MC.axZ;
	fbXlhMotionAxisZ.pAxis         := ADR(z_axis);
	fbXlhMotionAxisZ.pbEs          := ADR(io.motion.bAxZsw);

	fbXlhMotionAxisC.fbAxisPlcOpen REF= MC.axC;
	fbXlhMotionAxisC.pAxis         := ADR(c_axis);

	motion.pfbXlhMotionAxis[1] := ADR(fbXlhMotionAxisX);
	motion.pfbXlhMotionAxis[2] := ADR(fbXlhMotionAxisY);
	motion.pfbXlhMotionAxis[3] := ADR(fbXlhMotionAxisZ);
	motion.pfbXlhMotionAxis[4] := ADR(fbXlhMotionAxisC);
END_IF

IF bMagnet THEN
	motion.uiMagnetDutyCycle := uiMAGNET_ON;
ELSE
	motion.uiMagnetDutyCycle := uiMAGNET_OFF;
END_IF

METHOD read : BOOL
VAR_INPUT
END_VAR
gpio.read();
terminal.read();
motion.read();
END_METHOD

METHOD write : BOOL
VAR_INPUT
END_VAR
gpio.write();
terminal.write();
motion.write();
END_METHOD

END_PROGRAM

// xLH_base/app/MC
PROGRAM MC
VAR
	iState: INT;
	iHomingState: INT;
	
	fbPickAndPlace: FB_AXG_PICK_AND_PLACE;
	fbAxGmr: FB_AXG_MOVE_RELATIVE;
	fbAxGma: FB_AXG_MOVE_ABSOLUTE;
	
	axX: FB_PLC_OPEN_AXIS := (fVel:=fVEL, fAcc:=fACC_DEC, fDec:=fACC_DEC, fJerk:=fJERK);
	axY: FB_PLC_OPEN_AXIS := (fVel:=fVEL, fAcc:=fACC_DEC, fDec:=fACC_DEC, fJerk:=fJERK);
	axZ: FB_PLC_OPEN_AXIS := (fVel:=fVEL, fAcc:=fACC_DEC, fDec:=fACC_DEC, fJerk:=fJERK);
	axC: FB_PLC_OPEN_AXIS := (fVel:=fVEL, fAcc:=fACC_DEC, fDec:=fACC_DEC, fJerk:=fJERK);	

	baxGenable: BOOL;
	mcAxGenable : MC_GroupEnable;
	mcAxGdisable : MC_GroupDisable;
	mcAxGreset: MC_GroupReset;
	mcAxGsetCoord : MC_SetCoordinateTransform;	
	mcAxGmla: MC_MoveLinearAbsolute := (Velocity := fVEL, Acceleration := fACC_DEC, Deceleration := fACC_DEC, Jerk := fJERK);
	mcAxGmlr: MC_MoveLinearRelative := (Velocity := fVEL, Acceleration := fACC_DEC, Deceleration := fACC_DEC, Jerk := fJERK);	
	mcAxGcoordRef : MC_COORD_REF;
	bStartup: BOOL := TRUE;
	
	bCnc: BOOL;
	bError: BOOL;
END_VAR
VAR CONSTANT
	// Motion profile
	fVEL : LREAL := 30.0;
	fVEL_HOMING : LREAL := 2.0;
	fACC_DEC : LREAL := 20.0;
	fJERK : LREAL := 100.0;	
	
	// Homing
	fHOMING_FAST_FACTOR : LREAL :=  3.0;
	fHOMING_OFFSET_X    : LREAL := -5.0;
	fHOMING_OFFSET_Y    : LREAL := -5.0;
	fHOMING_OFFSET_Z    : LREAL := -5.0;
	
	// State constants (main state machine)
	STATE_STARTUP        : INT :=    0;
	STATE_HOMING         : INT :=   50;
	STATE_PRE_CMD        : INT :=  130;
	STATE_INIT_DONE      : INT := 999;
	STATE_RESET_CMDS     : INT := 1000;
	STATE_WAIT_CMD       : INT := 1010;
	STATE_MANUAL_MODE    : INT := 2000;
	STATE_PNP_CONVEYOR   : INT := 3000;
	STATE_APP_SQUARE_MODE: INT := 3100;
	STATE_CNC_MODE       : INT := 4000;
	STATE_ERROR          : INT := 9000;

	// Sub-states for the homing action
	STATE_POWER          : INT :=   50;
	STATE_DISABLE_GROUP  : INT :=  100;
	STATE_HOMING_ZA      : INT :=  110;
	STATE_HOMING_XY      : INT :=  115;
	STATE_ENABLE_GROUP   : INT :=  120;
END_VAR

IF bStartup THEN
	bStartup := FALSE;
	axInitPointers();
END_IF

read_io();

fbAxGmr();
fbAxGma();
fbPickAndPlace();
MANUAL_MODE(bEnable:=((iState = STATE_WAIT_CMD) OR (iState = STATE_MANUAL_MODE)));
APP_SQUARE_MODE(bEnable:=((iState = STATE_WAIT_CMD) OR (iState = STATE_APP_SQUARE_MODE)));
CNC_MODE(bEnable:=((iState = STATE_WAIT_CMD) OR (iState = STATE_CNC_MODE)));

IF bError THEN
	iState := STATE_ERROR;
END_IF

CASE iState OF
	// ============================================================================================
	// STARTUP AND INITIALIZATION
	// ============================================================================================
	
	// Initial state: clear all FB Execute flags, then run the homing sequence
	STATE_STARTUP:
		axSmExecuteToFalse();
		axGexecuteToFalse();		
		fbPickAndPlace.bExecute := FALSE;
		iHomingState := STATE_POWER;
		iState := STATE_HOMING;

	// Power axes, disable group, home Z/A then X/Y, re-enable group (see homing action)
	STATE_HOMING:
		homing();

	// Clear all Execute flags before the command cycle (clean transition)
	STATE_PRE_CMD:
		axSmExecuteToFalse();	
		axGexecuteToFalse();	
		fbPickAndPlace.bExecute := FALSE;
		iState := STATE_RESET_CMDS;
	
	

	// ============================================================================================
	// Commands
	// ============================================================================================
	
	// Reset command parameters (Vel/Acc/Jerk) and switch to the wait state
	STATE_RESET_CMDS:
		axCmdReset();
		axSmExecuteToFalse();
		axGexecuteToFalse();		
		iState := STATE_INIT_DONE;
		
	STATE_INIT_DONE:
		iState := STATE_WAIT_CMD;
		
	// Wait for operator input: evaluate jog buttons, auto PNP or CNC trigger
	STATE_WAIT_CMD:
		IF MANUAL_MODE.iState > MANUAL_MODE.STATE_IDLE THEN iState := STATE_MANUAL_MODE; END_IF
		IF APP_SQUARE_MODE.iState > APP_SQUARE_MODE.STATE_IDLE THEN iState := STATE_APP_SQUARE_MODE; END_IF
		IF CNC_MODE.iState > CNC_MODE.STATE_IDLE  THEN iState := STATE_CNC_MODE; END_IF
		IF io.terminal.bF3 THEN iState := STATE_STARTUP; END_IF

	// ============================================================================================
	// Axis jog mode (delegated to MANUAL_MODE program)
	// ============================================================================================

	// Run the MANUAL_MODE state machine until it returns to its idle state
	STATE_MANUAL_MODE:
		IF MANUAL_MODE.iState = MANUAL_MODE.STATE_IDLE THEN
			iState := STATE_RESET_CMDS;
		END_IF

	// ============================================================================================
	// Pick and Place
	// ============================================================================================

	STATE_PNP_CONVEYOR:
		;

	// Run the APP_SQUARE_MODE state machine until it returns to its idle state
	STATE_APP_SQUARE_MODE:
		IF APP_SQUARE_MODE.iState = APP_SQUARE_MODE.STATE_IDLE THEN
			iState := STATE_RESET_CMDS;
		END_IF

	// ============================================================================================
	// CNC Interpolation (delegated to CNC_MODE program)
	// ============================================================================================

	// CNC_MODE() is invoked cyclically from the program body; just monitor its state here
	STATE_CNC_MODE:
		IF CNC_MODE.iState = CNC_MODE.STATE_IDLE THEN
			iState := STATE_RESET_CMDS;
		END_IF

	// ============================================================================================
	// Error handling
	// ============================================================================================

	// Error state: halt all FBs and wait for bError to be acknowledged
	STATE_ERROR:
		axSmExecuteToFalse();
		axGexecuteToFalse();
		fbPickAndPlace.bExecute := FALSE;
		IF NOT bError THEN
			iState := STATE_RESET_CMDS;
		END_IF

END_CASE

write_io();

ACTION write_io:
// RGB Visualisierung

IF iState < STATE_INIT_DONE THEN
	io.terminal.eRgbReset := RGB.RED;
ELSE
	io.terminal.eRgbReset := RGB.OFF;
END_IF

IF MANUAL_MODE.iState > MANUAL_MODE.STATE_IDLE THEN
	IF MANUAL_MODE.iState > MANUAL_MODE.STATE_WAIT_CMD THEN
		io.terminal.eRgbManual := RGB.BLUE;
	ELSE
		io.terminal.eRgbManual := RGB.GREEN;
	END_IF
	io.terminal.eRgbAxEncoderC := RGB.GREEN;
	io.terminal.eRgbAxEncoderXY := RGB.GREEN;
	io.terminal.eRgbAxEncoderZ := RGB.GREEN;
ELSE
	io.terminal.eRgbManual := RGB.OFF;
	io.terminal.eRgbAxEncoderC := RGB.OFF;
	io.terminal.eRgbAxEncoderXY := RGB.OFF;
	io.terminal.eRgbAxEncoderZ := RGB.OFF;
END_IF

IF APP_SQUARE_MODE.iState > APP_SQUARE_MODE.STATE_IDLE THEN
	io.terminal.eRgbF1 := RGB.GREEN;
ELSE
	io.terminal.eRgbF1 := RGB.OFF;
END_IF

IF CNC_MODE.iState > CNC_MODE.STATE_IDLE THEN
	io.terminal.eRgbF2 := RGB.GREEN;
ELSE
	io.terminal.eRgbF2 := RGB.OFF;
END_IF

IF io.motion.uiMagnetDutyCycle > 0 THEN
	io.terminal.eRgbMagnet := RGB.GREEN;
ELSE
	io.terminal.eRgbMagnet := RGB.OFF;
END_IF

IF io.terminal.rVelMaster <= 0.1 THEN
	io.terminal.eRgbVelMaster := RGB.RED;
ELSIF (io.terminal.rVelMaster > 0.1) AND (io.terminal.rVelMaster <= 0.9) THEN
	io.terminal.eRgbVelMaster := RGB.GREEN;
ELSIF io.terminal.rVelMaster > 0.9 THEN
	io.terminal.eRgbVelMaster := RGB.BLUE;
ELSE
	io.terminal.eRgbVelMaster := RGB.OFF;
END_IF

io.write();
END_ACTION

ACTION read_io:
io.read();
END_ACTION

ACTION axSmExecuteToFalse:
axX.executeToFalse();
axY.executeToFalse();
axZ.executeToFalse();
axC.executeToFalse();
END_ACTION

ACTION axGexecuteToFalse:
mcAxGenable(AxisGroup := AxisGroup, Execute := FALSE);
mcAxGdisable(AxisGroup := AxisGroup, Execute := FALSE);
mcAxGreset(AxisGroup := AxisGroup, Execute := FALSE);
mcAxGsetCoord(AxisGroup := AxisGroup, Execute := FALSE);

fbAxGma.bExecute := FALSE;
fbAxGmr.bExecute := FALSE;
mcAxGmla(AxisGroup := AxisGroup, Execute := FALSE);
mcAxGmlr(AxisGroup := AxisGroup, Execute := FALSE);
END_ACTION

ACTION axInitPointers:
axX.pAxis := ADR(x_axis);
axY.pAxis := ADR(y_axis);
axZ.pAxis := ADR(z_axis);
axC.pAxis := ADR(c_axis);	

fbAxGmr.axGmr REF= mcAxGmlr;
fbAxGmr.axG REF= AxisGroup;  
fbAxGma.axGma REF= mcAxGmla;
fbAxGma.axG REF= AxisGroup;

fbPickAndPlace.fbAxisPlcOpenGma REF= fbAxGma;

MANUAL_MODE.fbAxGmr REF= fbAxGmr;
MANUAL_MODE.fbAxGma REF= fbAxGma;
APP_SQUARE_MODE.fbPickAndPlace REF= fbPickAndPlace;
CNC_MODE.fbAxGma REF= fbAxGma;
END_ACTION

ACTION axPowerOn:
axX.mcp.Enable := TRUE; axX.mcp.bRegulatorOn := TRUE; axX.mcp.bDriveStart := TRUE;
axY.mcp.Enable := TRUE; axY.mcp.bRegulatorOn := TRUE; axY.mcp.bDriveStart := TRUE;
axZ.mcp.Enable := TRUE; axZ.mcp.bRegulatorOn := TRUE; axZ.mcp.bDriveStart := TRUE;
axC.mcp.Enable := TRUE; axC.mcp.bRegulatorOn := TRUE; axC.mcp.bDriveStart := TRUE;
END_ACTION

ACTION axStartHomingZA:
io.fbXlhMotionAxisZ.fVelHoming         := fVEL_HOMING;
io.fbXlhMotionAxisZ.fVelHomingFast     := fHOMING_FAST_FACTOR * fVEL_HOMING;
io.fbXlhMotionAxisZ.eMcHomingDirection := MC_DIRECTION.positive;
io.fbXlhMotionAxisZ.fOffset            := fHOMING_OFFSET_Z;
io.fbXlhMotionAxisZ.bHoming            := TRUE;

io.fbXlhMotionAxisC.fVelHoming         := fVEL_HOMING;
io.fbXlhMotionAxisC.eMcHomingDirection := MC_DIRECTION.positive;
io.fbXlhMotionAxisC.bHoming            := TRUE;
END_ACTION

ACTION axStopHoming:
io.fbXlhMotionAxisX.bHoming := FALSE;
io.fbXlhMotionAxisY.bHoming := FALSE;
io.fbXlhMotionAxisZ.bHoming := FALSE;
io.fbXlhMotionAxisC.bHoming := FALSE;
END_ACTION

ACTION axCmdReset:
axX.fVel := fVEL; axX.fAcc := fACC_DEC; axX.fJerk := fJERK;
axY.fVel := fVEL; axY.fAcc := fACC_DEC; axY.fJerk := fJERK;
axZ.fVel := fVEL; axZ.fAcc := fACC_DEC; axZ.fJerk := fJERK;
END_ACTION

ACTION axSetDefaultKinValues:
io.fbXlhMotionAxisX.fbAxisPlcOpen.fVel := fVEL;
io.fbXlhMotionAxisX.fbAxisPlcOpen.fAcc := fACC_DEC;
io.fbXlhMotionAxisX.fbAxisPlcOpen.fDec := fACC_DEC;
io.fbXlhMotionAxisX.fbAxisPlcOpen.fJerk := fJERK;

io.fbXlhMotionAxisY.fbAxisPlcOpen.fVel := fVEL;
io.fbXlhMotionAxisY.fbAxisPlcOpen.fAcc := fACC_DEC;
io.fbXlhMotionAxisY.fbAxisPlcOpen.fDec := fACC_DEC;
io.fbXlhMotionAxisY.fbAxisPlcOpen.fJerk := fJERK;

io.fbXlhMotionAxisZ.fbAxisPlcOpen.fVel := fVEL;
io.fbXlhMotionAxisZ.fbAxisPlcOpen.fAcc := fACC_DEC;
io.fbXlhMotionAxisZ.fbAxisPlcOpen.fDec := fACC_DEC;
io.fbXlhMotionAxisZ.fbAxisPlcOpen.fJerk := fJERK;

io.fbXlhMotionAxisC.fbAxisPlcOpen.fVel := fVEL;
io.fbXlhMotionAxisC.fbAxisPlcOpen.fAcc := fACC_DEC;
io.fbXlhMotionAxisC.fbAxisPlcOpen.fDec := fACC_DEC;
io.fbXlhMotionAxisC.fbAxisPlcOpen.fJerk := fJERK;
END_ACTION

ACTION axStartHomingXY:
io.fbXlhMotionAxisX.fVelHoming         := fVEL_HOMING;
io.fbXlhMotionAxisX.fVelHomingFast     := fHOMING_FAST_FACTOR * fVEL_HOMING;
io.fbXlhMotionAxisX.eMcHomingDirection := MC_DIRECTION.positive;
io.fbXlhMotionAxisX.fOffset            := fHOMING_OFFSET_X;
io.fbXlhMotionAxisX.bHoming            := TRUE;

io.fbXlhMotionAxisY.fVelHoming         := fVEL_HOMING;
io.fbXlhMotionAxisY.fVelHomingFast     := fHOMING_FAST_FACTOR * fVEL_HOMING;
io.fbXlhMotionAxisY.eMcHomingDirection := MC_DIRECTION.positive;
io.fbXlhMotionAxisY.fOffset            := fHOMING_OFFSET_Y;
io.fbXlhMotionAxisY.bHoming            := TRUE;
END_ACTION

ACTION homing:
CASE iHomingState OF
	// Power up the axes and wait until all four are in the "Standstill" state
	STATE_POWER:
		axPowerOn();
		// https://content.helpme-codesys.com/en/libs/SM3_Basic/Current/SM3_Basic/DataTypes/DriveInterface/SMC_AXIS_STATE.html
		IF (axX.mcp.Status AND x_axis.nAxisState = SMC_AXIS_STATE.standstill) AND
		   (axY.mcp.Status AND y_axis.nAxisState = SMC_AXIS_STATE.standstill) AND
		   (axZ.mcp.Status AND z_axis.nAxisState = SMC_AXIS_STATE.standstill) AND
		   (axC.mcp.Status AND c_axis.nAxisState = SMC_AXIS_STATE.standstill) THEN
			axSmExecuteToFalse();
			iHomingState := STATE_DISABLE_GROUP;
		END_IF

	// Disable the axis group before homing (homing requires per-axis control)
	STATE_DISABLE_GROUP:
		IF baxGenable THEN
			mcAxGdisable(AxisGroup := AxisGroup, Execute := TRUE);
			IF mcAxGdisable.Done THEN
				baxGenable := FALSE;
				axGexecuteToFalse();
				iHomingState := STATE_HOMING_ZA;
			END_IF
		ELSE
			iHomingState := STATE_HOMING_ZA;
		END_IF

	// Phase 1: start homing for axes Z and A and wait for completion
	STATE_HOMING_ZA:
		axStartHomingZA();
		IF io.fbXlhMotionAxisZ.bHomingDone AND
		   io.fbXlhMotionAxisC.bHomingDone THEN
			axSmExecuteToFalse();
			iHomingState := STATE_HOMING_XY;
		END_IF

	// Phase 2: start homing for axes X and Y and wait for completion
	STATE_HOMING_XY:
		axStartHomingXY();
		IF io.fbXlhMotionAxisX.bHomingDone AND
		   io.fbXlhMotionAxisY.bHomingDone THEN
			axSmExecuteToFalse();
			axStopHoming();
			axSetDefaultKinValues();
			iHomingState := STATE_ENABLE_GROUP;
		END_IF

	// Re-enable the axis group after successful homing
	STATE_ENABLE_GROUP:
		IF NOT baxGenable THEN
			mcAxGenable(AxisGroup := AxisGroup, Execute := TRUE);
			IF mcAxGenable.Done THEN
				baxGenable := TRUE;
				axGexecuteToFalse();
				iState := STATE_PRE_CMD;
			END_IF
		ELSE
			iState := STATE_PRE_CMD;
		END_IF
END_CASE
END_ACTION

END_PROGRAM

// xLH_base/app/MANUAL_MODE
// =====================================================================
// MANUAL_MODE
// Manual jog state machine, called from MC when iState = STATE_
// MC sets the target (smcPosRef for the XYZ group, mcmr.Distance for the
// A axis) and selects the sub-state (STATE_STEP_REL / STATE_STEP_ABS /
// STATE_STEP_REL_A / STATE_STEP_ABS_A). The case below executes the move
// and returns to STATE_WAIT_CMD on completion; MC reads STATE_WAIT_CMD as the
// "done" signal and returns to STATE_RESET_CMDS.
// =====================================================================
PROGRAM MANUAL_MODE
VAR_INPUT
	bEnable: BOOL;
	fbAxGmr: REFERENCE TO FB_AXG_MOVE_RELATIVE;
	fbAxGma: REFERENCE TO FB_AXG_MOVE_ABSOLUTE;
END_VAR
VAR_OUTPUT
	iState: INT;
END_VAR
VAR
	bXp: BOOL;
	bXm: BOOL;
	bYp: BOOL;
	bYm: BOOL;
	bZp: BOOL;
	bZm: BOOL;
	bCp: BOOL;
	bCm: BOOL;
	fStepXY: LREAL;
	fStepZ: LREAL;
	fStepC: LREAL;
	fStepOffsetXY: LREAL := 10.0;
	fStepOffsetZ: LREAL := 2.5;
	fStepOffsetC: LREAL := 50.0;
	
	smcPosRef: SMC_POS_REF;
	smcPosRef1 : SMC_POS_REF := (c:= (X:=-102.7, Y:=-46.1, Z:=-52.5));
	smcPosRef2 : SMC_POS_REF := (c:= (X:=-122.7, Y:=-66.1, Z:=-52.5));
	smcPosRef3 : SMC_POS_REF := (c:= (X:=-122.7, Y:=-66.1, Z:=-52.5));
	smcPosRef4 : SMC_POS_REF := (c:= (X:=-122.7, Y:=-66.1, Z:=-52.5));
	smcPosRef5 : SMC_POS_REF := (c:= (X:=-122.7, Y:=-66.1, Z:=-52.5));
	smcPosRef6 : SMC_POS_REF := (c:= (X:=-122.7, Y:=-66.1, Z:=-52.5));
	
END_VAR
VAR CONSTANT
	STATE_DISABLED  : INT := 	0;
	STATE_IDLE      : INT :=  500;
	STATE_INIT      : INT :=  700;
	STATE_WAIT_CMD  : int := 1000;
	STATE_STEP_REL   : INT := 2000;
	STATE_STEP_ABS   : INT := 2010;
	STATE_STEP_REL_A : INT := 2020;
	STATE_STEP_ABS_A : INT := 2030;
END_VAR

fStepC := LIMIT(1.0, fStepOffsetC + INT_TO_LREAL(io.terminal.iAxEncoderC) * 1.0, 100.0);
fStepXY := LIMIT(0.1, fStepOffsetXY + INT_TO_LREAL(io.terminal.iAxEncoderXY) * 0.1, 25.0);
fStepZ := LIMIT(0.1, fStepOffsetZ + INT_TO_LREAL(io.terminal.iAxEncoderZ) * 0.1, 10.0);

IF iState > STATE_INIT THEN
	IF io.terminal.bRtMagnet THEN
		io.bMagnet := NOT io.bMagnet;
	END_IF
ELSE
	;
END_IF


CASE iState OF
	STATE_DISABLED:
		IF bEnable THEN
			iState := STATE_IDLE;
		END_IF
		
	STATE_IDLE:
		IF NOT bEnable THEN
			iState := STATE_DISABLED;
		END_IF
		IF io.terminal.bRtManual THEN
			iState := STATE_INIT;
		END_IF
		
	STATE_INIT:
		iState := STATE_WAIT_CMD;
		
	STATE_WAIT_CMD:
		IF NOT bEnable THEN
			iState := STATE_DISABLED;
		END_IF
		
		IF io.terminal.bRtReset THEN
			iState := STATE_IDLE;
		END_IF
		
		IF bXp OR io.terminal.bRtAxXp THEN 
			smcPosRef.c.X :=  fStepXY; smcPosRef.c.Y :=  0.0;   smcPosRef.c.Z :=  0.0;   
			iState := STATE_STEP_REL; 
		END_IF
		IF bXm OR io.terminal.bRtAxXm THEN 
			smcPosRef.c.X := -fStepXY; smcPosRef.c.Y :=  0.0;   smcPosRef.c.Z :=  0.0;   
			iState := STATE_STEP_REL; 
		END_IF
		IF bYp OR io.terminal.bRtAxYp THEN 
			smcPosRef.c.X :=  0.0;   smcPosRef.c.Y :=  fStepXY; smcPosRef.c.Z :=  0.0;   
			iState := STATE_STEP_REL; 
		END_IF
		IF bYm OR io.terminal.bRtAxYm THEN 
			smcPosRef.c.X :=  0.0;   smcPosRef.c.Y := -fStepXY; smcPosRef.c.Z :=  0.0;   
			iState := STATE_STEP_REL; 
		END_IF
		IF bZp OR io.terminal.bRtAxZp THEN 
			smcPosRef.c.X :=  0.0;   smcPosRef.c.Y :=  0.0;   smcPosRef.c.Z := fStepZ; 
			iState := STATE_STEP_REL; 
		END_IF
		IF bZm OR io.terminal.bRtAxZm THEN 
			smcPosRef.c.X :=  0.0;   smcPosRef.c.Y :=  0.0;   smcPosRef.c.Z := -fStepZ; 
			iState := STATE_STEP_REL; 
		END_IF
		IF bCp OR io.terminal.bRtAxCp THEN 
			io.fbXlhMotionAxisC.fbAxisPlcOpen.mcmr.Distance :=  fStepC; 
			iState := STATE_STEP_REL_A; 
		END_IF
		IF bCm OR io.terminal.bRtAxCm THEN 
			io.fbXlhMotionAxisC.fbAxisPlcOpen.mcmr.Distance := -fStepC; 
			iState := STATE_STEP_REL_A; 
		END_IF
		IF io.terminal.bRt1 THEN 
			smcPosRef := smcPosRef1;
			iState := STATE_STEP_ABS; 
		END_IF
		IF io.terminal.bRt2 THEN 
			smcPosRef := smcPosRef2;
			iState := STATE_STEP_ABS; 
		END_IF
		IF io.terminal.bRt3 THEN 
			smcPosRef := smcPosRef3;
			iState := STATE_STEP_ABS; 
		END_IF
		IF io.terminal.bRt4 THEN 
			smcPosRef := smcPosRef4;
			iState := STATE_STEP_ABS; 
		END_IF
		IF io.terminal.bRt5 THEN 
			smcPosRef := smcPosRef5;
			iState := STATE_STEP_ABS; 
		END_IF
		IF io.terminal.bRt6 THEN 
			smcPosRef := smcPosRef6;
			iState := STATE_STEP_ABS; 
		END_IF


	// Relative axis-group jog by smcPosRef on the previously selected axis
	STATE_STEP_REL:
		fbAxGmr.bExecute := TRUE;
		fbAxGmr.tPosRef := smcPosRef;
		IF fbAxGmr.bDone THEN
			MC.axGexecuteToFalse();
			iState := STATE_WAIT_CMD;
		END_IF

	// Absolute axis-group move to the target position smcPosRef
	STATE_STEP_ABS:
		fbAxGma.bExecute := TRUE;
		fbAxGma.tPosRef := smcPosRef;
		IF fbAxGma.bDone THEN
			MC.axGexecuteToFalse();
			iState := STATE_WAIT_CMD;
		END_IF

	// Relative move on the A axis (uses the per-axis FB_PLC_OPEN_AXIS)
	STATE_STEP_REL_A:
		io.fbXlhMotionAxisC.fbAxisPlcOpen.mcmr.Execute := TRUE;
		IF io.fbXlhMotionAxisC.fbAxisPlcOpen.mcmr.Done THEN
			io.fbXlhMotionAxisC.fbAxisPlcOpen.executeToFalse();
			iState := STATE_WAIT_CMD;
		END_IF
END_CASE

ACTION TODO:
(*
ToDo
- Reset Encoder via CANopen
- Umschaltung JOG STEP mit Visu RGB
- Definition von Punktreferenzen
*)
END_ACTION

END_PROGRAM

// xLH_base/app/MOTION_BASE/FB_PLC_OPEN_AXIS
// =====================================================================
// FB_PLC_OPEN_AXIS
// Bundles the PLCopen motion blocks (MC_Power, MC_Stop, MC_MoveAbsolute,
// MC_MoveRelative, MC_MoveVelocity, MC_Reset, MC_ReadStatus,
// MC_ReadAxisError, SMC_ReadFBError) for a single axis.
// Manages default values for velocity/acceleration/jerk, provides
// actual values (fActPos/fActVel/fActAcc) and aggregates MC errors into
// bError. Action plcOpen() invokes all MC blocks cyclically, action
// executeToFalse() clears the Execute flags.
// =====================================================================
FUNCTION_BLOCK FB_PLC_OPEN_AXIS
VAR_INPUT	
	fVel: LREAL := 200.0;
	fAcc: LREAL := 750.0;
	fDec: LREAL := 750.0;
	fJerk: LREAL := 10000.0;
	
	mcrs: MC_ReadStatus := (Enable:=TRUE);
	mcrae: MC_ReadAxisError := (Enable:=TRUE);
	mcr: MC_Reset;
	smcrfbe: SMC_ReadFBError;
	mcp: MC_Power := (Enable:=FALSE, bRegulatorOn:=FALSE, bDriveStart:=FALSE);
	mcs: MC_Stop;
	mcma: MC_MoveAbsolute := (Velocity:=100.0, Acceleration:=1000.0, Deceleration:=1000.0, Jerk:=10000.0);
	mcmr: MC_MoveRelative := (Velocity:=100.0, Acceleration:=1000.0, Deceleration:=1000.0, Jerk:=10000.0);
	mcmv: MC_MoveVelocity := (Velocity:=100.0, Acceleration:=1000.0, Deceleration:=1000.0, Jerk:=10000.0, Direction:=-1);// 1 positive, -1 negative
	
	pAxis: POINTER TO AXIS_REF_SM3; 
	// https://content.helpme-codesys.com/en/libs/SM3_Drive_PosControl/Current/AXIS_REF_POSCONTROL.html
	//axisPosControl: REFERENCE TO AXIS_REF_POSCONTROL;
END_VAR
VAR_OUTPUT	
	bError: BOOL;
	fActPos: LREAL;
	fActVel: LREAL;
	fActAcc: LREAL;
END_VAR
VAR
END_VAR

// Call the PLCopen motion blocks
plcOpen();

// Error evaluation
bError := mcs.Error OR mcmr.Error OR mcma.Error OR mcmv.Error;

// Assign motion control actual values
IF pAxis > 16#0 THEN
	fActPos := pAxis^.fActPosition;
	fActVel := pAxis^.fActVelocity;
	fActAcc := pAxis^.fActAcceleration;
END_IF

ACTION plcOpen:
IF pAxis > 16#0 THEN
	// Call the PLCopen motion control blocks
	mcrs(Axis:=pAxis^);// MC_ReadStatus https://help.codesys.com/search;version=3.5.17.0;term=MC_ReadStatus
	mcrae(Axis:=pAxis^);// MC_ReadAxisError https://help.codesys.com/webapp/ML6Svtks37sht2hVC_6YLIhf2ZY%2FMC_ReadAxisError;product=SM3_Basic;version=4.9.0.0
	mcr(Axis:=pAxis^);// MC_Reset https://help.codesys.com/webapp/xiNnxNPAb5nA4ocm6PFB_cHgUb4%2FMC_Reset;product=SM3_Basic;version=4.9.0.0
	smcrfbe(Axis:=pAxis^);// SMC_ReadFBError https://help.codesys.com/webapp/xUeuGLdUseEDKMLaPLQmdZO45P8%2FSMC_ReadFBError;product=SM3_Basic;version=4.9.0.0
	mcp(Axis:=pAxis^);// MC_Power https://help.codesys.com/webapp/xiNnxNPAb5nA4ocm6PFB_cHgUb4%2FMC_Power;product=SM3_Basic;version=4.9.0.0
	//mch(Axis:=pAxis^);// MC_Home https://content.helpme-codesys.com/en/libs/SM3_Basic/Current/SM3_Basic/POUs/Movement/MC_Home.html
	
	mcs.Deceleration := fDec;
	mcs.Jerk := fJerk;
	mcs(Axis:=pAxis^);// MC_Stop https://help.codesys.com/webapp/xUeuGLdUseEDKMLaPLQmdZO45P8%2FSMC_ReadFBError;product=SM3_Basic;version=4.9.0.0
	
	mcma.Velocity := fVel;
	mcma.Acceleration := fAcc;
	mcma.Deceleration := fDec;
	mcma.Jerk := fJerk;
	mcma(Axis:=pAxis^);// MC_MoveAbsolute https://help.codesys.com/webapp/74YgxSD47ycAkED81whSoB9i6wQ%2FMC_MoveAbsolute;product=SM3_Basic;version=4.9.0.0
	
	mcmr.Velocity := fVel;
	mcmr.Acceleration := fAcc;
	mcmr.Deceleration := fDec;
	mcmr.Jerk := fJerk;
	mcmr(Axis:=pAxis^);// MC_MoveRelative https://help.codesys.com/webapp/74YgxSD47ycAkED81whSoB9i6wQ%2FMC_MoveRelative;product=SM3_Basic;version=4.9.0.0
	
	mcmv.Velocity := fVel;
	mcmv.Acceleration := fAcc;
	mcmv.Deceleration := fDec;
	mcmv.Jerk := fJerk;
	mcmv(Axis:=pAxis^);// MC_MoveVelocity https://help.codesys.com/webapp/74YgxSD47ycAkED81whSoB9i6wQ%2FMC_MoveVelocity;product=SM3_Basic;version=4.9.0.0
	
	// SoftMotion: https://help.codesys.com/webapp/_sm_components;product=codesys_softmotion;version=4.10.0.0
	// Drive: https://help.codesys.com/webapp/_sm_inserting_connected_drive_devices;product=codesys_softmotion;version=4.10.0.0
	// SMC Error: https://help.codesys.com/webapp/4icXWiTEEU7jfvlz7ATrx-Bu-fs%2FSMC_ERROR;product=SM3_Basic;version=4.0.0.0
END_IF
END_ACTION

ACTION executeToFalse:
mcr.Execute := FALSE;
mcs.Execute := FALSE;
mcma.Execute := FALSE;
mcmr.Execute := FALSE;
mcmv.Execute := FALSE;
END_ACTION

END_FUNCTION_BLOCK

// xLH_base/app/MOTION_BASE/FB_AXG_MOVE_RELATIVE
// =====================================================================
// FB_AXG_MOVE_RELATIVE
// Wrapper around MC_MoveLinearRelative (axis-group motion). Identical
// to FB_AXG_MOVE_ABSOLUTE, but with a relative distance tPosRef instead
// of an absolute target position. Default parameters such as
// BlendingHigh, TMCornerDistance and MCS are hard-coded.
// =====================================================================
FUNCTION_BLOCK FB_AXG_MOVE_RELATIVE
VAR_INPUT
	bExecute: BOOL;
	tPosRef: SMC_POS_REF;
	axGmr: REFERENCE TO MC_MoveLinearRelative;
	axG: REFERENCE TO AXIS_GROUP_REF_SM3;
END_VAR
VAR_OUTPUT
	bDone: BOOL;
END_VAR
VAR CONSTANT
	fCORNER_DISTANCE : LREAL := 50.0;
END_VAR

axGmr.Execute := bExecute;
axGmr.Distance := tPosRef;
axGmr.BufferMode := MC_BUFFER_MODE.BlendingHigh;
axGmr.TransitionMode := MC_TRANSITION_MODE.TMCornerDistance;
axGmr.TransitionParameter[0] := fCORNER_DISTANCE;
axGmr.CoordSystem := SMC_COORD_SYSTEM.MCS;
axGmr(AxisGroup := axG);
bDone := axGmr.Done;

END_FUNCTION_BLOCK

// xLH_base/app/MOTION_BASE/FB_AXG_MOVE_ABSOLUTE
// =====================================================================
// FB_AXG_MOVE_ABSOLUTE
// Wrapper around MC_MoveLinearAbsolute (axis-group motion). Sets fixed
// default parameters (BufferMode = BlendingHigh, TransitionMode =
// TMCornerDistance with fCORNER_DISTANCE, CoordSystem = MCS) and
// forwards bExecute/tPosRef and bDone to/from the SoftMotion group.
// =====================================================================
FUNCTION_BLOCK FB_AXG_MOVE_ABSOLUTE
VAR_INPUT
	bExecute: BOOL;
	tPosRef: SMC_POS_REF;
	axGma: REFERENCE TO MC_MoveLinearAbsolute;
	axG: REFERENCE TO AXIS_GROUP_REF_SM3;
END_VAR
VAR_OUTPUT
	bDone: BOOL;
END_VAR
VAR CONSTANT
	fCORNER_DISTANCE : LREAL := 50.0;
END_VAR

axGma.Execute := bExecute;
axGma.Position := tPosRef;
axGma.BufferMode := MC_BUFFER_MODE.BlendingHigh;
axGma.TransitionMode := MC_TRANSITION_MODE.TMCornerDistance;
axGma.TransitionParameter[0] := fCORNER_DISTANCE;
axGma.CoordSystem := SMC_COORD_SYSTEM.MCS;
axGma(AxisGroup := axG);
bDone := axGma.Done;

END_FUNCTION_BLOCK

// xLH_base/app/APP_SQUARE_MODE
// =====================================================================
// APP_SQUARE_MODE
// Pick-and-place square application with the FB_PNP_SQUARE sequencer
// integrated directly. On a 2D grid, 5 steps from the inner square
// (PNP_STEPS) are run in combination with 4 outer grid points
// (PNP_GRID); each iteration drives MC.fbPickAndPlace.
//   - inner counter iI iterates 0..3 (grid points)
//   - outer counter iN iterates 0..4 (square steps)
//   - MC.bAuto = TRUE restarts the sequence endlessly; MC.bAuto =
//     FALSE returns to STATE_IDLE after one complete round.
// io.bMagnet is forwarded from MC.fbPickAndPlace.bMagnet on every
// cycle the program runs. MC reads STATE_IDLE as the "done" signal.
// =====================================================================
PROGRAM APP_SQUARE_MODE
VAR_INPUT
	bEnable: BOOL;
	fbPickAndPlace: REFERENCE TO FB_AXG_PICK_AND_PLACE;
END_VAR
VAR_OUTPUT
	iState : INT;
END_VAR
VAR
	POS_REF : SMC_POS_REF := (c:= (X:=-122.7, Y:=-66.1, Z:=-52.5));
	iN     : INT;
	iI     : INT;
	bStart: BOOL;
END_VAR
VAR CONSTANT
	STATE_DISABLED      : INT :=    0;
	STATE_IDLE          : INT :=  500;
	STATE_PNP_INIT      : INT := 3100;
	STATE_PNP_EXECUTE   : INT := 3110;
	STATE_PNP_INNER_INC : INT := 3120;
	STATE_PNP_OUTER_INC : INT := 3130;
	STATE_PNP_LOOP      : INT := 3140;

	iPNP_OUTER_COUNT : INT := 5;
	PNP_STEPS : ARRAY[0..4] OF ST_PnpStep := [
		(fPickX:=  0.0, fPickY:=  0.0, fPlaceX:= 20.0, fPlaceY:= 20.0),
		(fPickX:= 20.0, fPickY:= 20.0, fPlaceX:= 20.0, fPlaceY:=-20.0),
		(fPickX:= 20.0, fPickY:=-20.0, fPlaceX:=-20.0, fPlaceY:=-20.0),
		(fPickX:=-20.0, fPickY:=-20.0, fPlaceX:=-20.0, fPlaceY:= 20.0),
		(fPickX:=-20.0, fPickY:= 20.0, fPlaceX:=  0.0, fPlaceY:=  0.0)
	];

	iPNP_INNER_COUNT : INT := 2;
	PNP_GRID : ARRAY[0..1] OF ST_PnpStep := [
		(fPickX:= 0.0, fPickY:=  0.0),
		(fPickX:= 0.0, fPickY:= -70.0)
	];
END_VAR

// Forward magnet state from the pick-and-place FB to the io layer
IF iState > STATE_DISABLED THEN
	io.bMagnet := fbPickAndPlace.bMagnet;
END_IF

CASE iState OF
	STATE_DISABLED:
		IF bEnable THEN
			iState := STATE_IDLE;
		END_IF
	
	STATE_IDLE:
		IF NOT bEnable THEN
			iState := STATE_DISABLED;
		END_IF
		fbPickAndPlace.bExecute := FALSE;
		IF bStart OR io.terminal.bF1 THEN 
			iState := STATE_PNP_INIT; 
		END_IF 

	// Initialise inner/outer counters before the first iteration
	STATE_PNP_INIT:
		iI := 0;
		iN := 0;
		iState := STATE_PNP_EXECUTE;

	// Drive fbPickAndPlace with the current pick/place targets
	STATE_PNP_EXECUTE:
		fbPickAndPlace.tPosPick.c.X  := POS_REF.c.X + PNP_STEPS[iN].fPickX  + PNP_GRID[iI].fPickX;
		fbPickAndPlace.tPosPick.c.Y  := POS_REF.c.Y + PNP_STEPS[iN].fPickY  + PNP_GRID[iI].fPickY;
		fbPickAndPlace.tPosPick.c.Z  := POS_REF.c.Z;
		fbPickAndPlace.tPosPlace.c.X := POS_REF.c.X + PNP_STEPS[iN].fPlaceX + PNP_GRID[iI].fPickX;
		fbPickAndPlace.tPosPlace.c.Y := POS_REF.c.Y + PNP_STEPS[iN].fPlaceY + PNP_GRID[iI].fPickY;
		fbPickAndPlace.tPosPlace.c.Z := POS_REF.c.Z;
		fbPickAndPlace.bExecute := TRUE;
		IF fbPickAndPlace.bDone THEN
			fbPickAndPlace.bExecute := FALSE;
			iState := STATE_PNP_INNER_INC;
		END_IF

	STATE_PNP_INNER_INC:
		iI := iI + 1;
		IF iI >= iPNP_INNER_COUNT THEN
			iI := 0;
			iState := STATE_PNP_OUTER_INC;
		ELSE
			iState := STATE_PNP_EXECUTE;
		END_IF

	STATE_PNP_OUTER_INC:
		iN := iN + 1;
		IF iN >= iPNP_OUTER_COUNT THEN
			iN := 0;
			iState := STATE_PNP_LOOP;
		ELSE
			iState := STATE_PNP_EXECUTE;
		END_IF

	// One complete round done: restart in auto mode, otherwise return to idle
	STATE_PNP_LOOP:
		IF bStart THEN
			iState := STATE_PNP_INIT;
		ELSE
			MC.axGexecuteToFalse();
			iState := STATE_IDLE;
		END_IF
END_CASE

END_PROGRAM

// xLH_base/app/MOTION_BASE/FB_AXG_PICK_AND_PLACE
// =====================================================================
// FB_AXG_PICK_AND_PLACE
// State machine for a pick-and-place sequence:
//   PICK_HOVER  -> move above the pick position to OFFSET_Z
//   PICK_DOWN   -> lower onto the pick position (Z = 0)
//   MAGNET_ON   -> activate magnet, wait T_MAGNET
//   PICK_LIFT   -> lift back to OFFSET_Z
//   PLACE_HOVER -> move above the place position to OFFSET_Z
//   PLACE_DOWN  -> lower onto the place position
//   MAGNET_OFF  -> deactivate magnet, wait T_MAGNET
//   PLACE_LIFT  -> lift back to OFFSET_Z
//   DONE        -> bDone := TRUE
// Uses the externally referenced FB_AXG_MOVE_ABSOLUTE (fbAxisPlcOpenGma) for the
// motions and exposes the magnet control output bMagnet.
// =====================================================================
FUNCTION_BLOCK FB_AXG_PICK_AND_PLACE
VAR_INPUT
	bExecute: BOOL;
	tPosPick: SMC_POS_REF;
	tPosPlace: SMC_POS_REF;
	fbAxisPlcOpenGma: REFERENCE TO FB_AXG_MOVE_ABSOLUTE;
END_VAR
VAR_OUTPUT
	iState: INT := 0;
	bDone: BOOL;
	bMagnet: BOOL;
END_VAR
VAR
	tonDelay1: TON;
END_VAR
VAR CONSTANT
	OFFSET_Z : LREAL := 10.0;
	T_MAGNET : TIME  := T#250MS;

	STATE_PICK_HOVER  : INT :=  0;
	STATE_PICK_DOWN   : INT := 10;
	STATE_MAGNET_ON   : INT := 20;
	STATE_PICK_LIFT   : INT := 30;
	STATE_PLACE_HOVER : INT := 40;
	STATE_PLACE_DOWN  : INT := 50;
	STATE_MAGNET_OFF  : INT := 60;
	STATE_PLACE_LIFT  : INT := 70;
	STATE_DONE        : INT := 80;
END_VAR

IF bExecute THEN
	CASE iState OF
		STATE_PICK_HOVER:  IF moveToOffset(tPosPick,  OFFSET_Z) THEN iState := STATE_PICK_DOWN;   END_IF
		STATE_PICK_DOWN:   IF moveToOffset(tPosPick,  0.0)      THEN iState := STATE_MAGNET_ON;   END_IF
		STATE_MAGNET_ON:   IF setMagnet(TRUE)                   THEN iState := STATE_PICK_LIFT;   END_IF
		STATE_PICK_LIFT:   IF moveToOffset(tPosPick,  OFFSET_Z) THEN iState := STATE_PLACE_HOVER; END_IF
		STATE_PLACE_HOVER: IF moveToOffset(tPosPlace, OFFSET_Z) THEN iState := STATE_PLACE_DOWN;  END_IF
		STATE_PLACE_DOWN:  IF moveToOffset(tPosPlace, 0.0)      THEN iState := STATE_MAGNET_OFF;  END_IF
		STATE_MAGNET_OFF:  IF setMagnet(FALSE)                  THEN iState := STATE_PLACE_LIFT;  END_IF
		STATE_PLACE_LIFT:  IF moveToOffset(tPosPlace, OFFSET_Z) THEN iState := STATE_DONE;        END_IF
		STATE_DONE:        bDone := TRUE;
	END_CASE
ELSE
	iState := STATE_PICK_HOVER;
	bMagnet := FALSE;
	bDone := FALSE;
END_IF

tonDelay1(IN := iState = STATE_MAGNET_ON OR iState = STATE_MAGNET_OFF, PT := T_MAGNET);

METHOD PRIVATE moveToOffset : BOOL
VAR_INPUT
	base    : SMC_POS_REF;
	zOffset : LREAL;
END_VAR
VAR
	target : SMC_POS_REF;
END_VAR
IF fbAxisPlcOpenGma.bDone THEN
	fbAxisPlcOpenGma.bExecute := FALSE;
	moveToOffset := TRUE;
ELSE
	target := base;
	target.c.Z := target.c.Z + zOffset;
	fbAxisPlcOpenGma.tPosRef := target;
	fbAxisPlcOpenGma.bExecute := TRUE;
END_IF
END_METHOD

METHOD PRIVATE setMagnet : BOOL
VAR_INPUT
	on : BOOL;
END_VAR
bMagnet := on;
setMagnet := tonDelay1.Q;
END_METHOD

END_FUNCTION_BLOCK

// xLH_base/app/CNC_MODE
// =====================================================================
// CNC_MODE
// CNC interpolation state machine with the SoftMotion chain integrated
// directly (formerly wrapped in FB_CNC_IPO):
//   SMC_CheckVelocities  -> validates/smooths the velocity profiles
//                           of the out-queue.
//   SMC_Interpolator     -> interpolates the path cyclically and
//                           provides the current setpoint piSetPosition.
//   SMC_ControlAxisByPos -> writes the per-axis setpoint directly to
//                           AXIS_REF_SM3 (X, Y, Z).
// On entry, the XYZ offsets are frozen so the G-code path starts
// relative to the current axis actual position.
// Called every cycle from MC.prg so the chain keeps ticking even
// when the program is in STATE_IDLE.
// =====================================================================
PROGRAM CNC_MODE
VAR_INPUT
	bEnable : BOOL;
	fbAxGma       : REFERENCE TO FB_AXG_MOVE_ABSOLUTE;
END_VAR
VAR_OUTPUT
	iState        : INT;
END_VAR
VAR
	POS_REF : SMC_POS_REF := (c:= (X:=-130.0, Y:=-75.0, Z:=-40.0));
	bExecute      : BOOL;
	poqDataIn     : POINTER TO SMC_OUTQUEUE;
	piSetPosition : SMC_POSINFO;
	fOffsetX      : LREAL;
	fOffsetY      : LREAL;
	fOffsetZ      : LREAL;
	bDone         : BOOL;
	bBusy         : BOOL;
	bError        : BOOL;
	wErrorID      : SMC_ERROR;

	fbCheckVel    : SMC_CheckVelocities;
	fbIpo         : SMC_Interpolator;
	fbCtrlX       : SMC_ControlAxisByPos;
	fbCtrlY       : SMC_ControlAxisByPos;
	fbCtrlZ       : SMC_ControlAxisByPos;
END_VAR
VAR CONSTANT
	STATE_DISABLED      : INT :=    0;
	STATE_IDLE          : INT :=  500;
	STATE_CNC_IPO_START : INT := 4000;
	STATE_CNC_IPO       : INT := 4010;

	dwIpoTime : DWORD := 4000;
END_VAR

// Cyclic interpolation chain (formerly FB_CNC_IPO body)
fbCheckVel(
	bExecute  := bExecute,
	poqDataIn := poqDataIn);

fbIpo(
	bExecute        := bExecute AND fbCheckVel.poqDataOut <> 0,
	poqDataIn       := fbCheckVel.poqDataOut,
	bSlow_Stop      := FALSE,
	bEmergency_Stop := FALSE,
	dOverride       := io.terminal.rVelMaster,
	dwIpoTime       := dwIpoTime,
	iVelMode        := TRAPEZOID);

piSetPosition := fbIpo.piSetPosition;

fbCtrlX(
	Axis         := x_axis,
	iStatus      := fbIpo.iStatus,
	bEnable      := bExecute,
	fSetPosition := fOffsetX + piSetPosition.dX);

fbCtrlY(
	Axis         := y_axis,
	iStatus      := fbIpo.iStatus,
	bEnable      := bExecute,
	fSetPosition := fOffsetY + piSetPosition.dY);

fbCtrlZ(
	Axis         := z_axis,
	iStatus      := fbIpo.iStatus,
	bEnable      := bExecute,
	fSetPosition := fOffsetZ + piSetPosition.dZ);

bDone  := fbIpo.bDone;
bBusy  := fbIpo.bBusy;
bError := fbCheckVel.bError OR fbIpo.bError OR fbCtrlX.bError OR fbCtrlY.bError OR fbCtrlZ.bError;

IF fbCheckVel.bError THEN
	wErrorID := fbCheckVel.wErrorID;
ELSIF fbIpo.bError THEN
	wErrorID := fbIpo.wErrorID;
ELSIF fbCtrlX.bError THEN
	wErrorID := fbCtrlX.iErrorID;
ELSIF fbCtrlY.bError THEN
	wErrorID := fbCtrlY.iErrorID;
ELSIF fbCtrlZ.bError THEN
	wErrorID := fbCtrlZ.iErrorID;
END_IF

// State machine
CASE iState OF
	STATE_DISABLED:
		IF bEnable THEN
			iState := STATE_IDLE;
		END_IF
	
	STATE_IDLE:
		IF NOT bEnable THEN
			iState := STATE_DISABLED;
		END_IF
		IF io.terminal.bRtF2 THEN
			iState := STATE_CNC_IPO_START;
		END_IF
		//bExecute := FALSE;

	// Move the XYZ axes to the reference point POS_REF before CNC interpolation
	STATE_CNC_IPO_START:
		fbAxGma.tPosRef := POS_REF;
		fbAxGma.bExecute := TRUE;
		IF fbAxGma.bDone THEN
			MC.axGexecuteToFalse();
			poqDataIn := ADR(DEMO_GCODE);
			// Freeze XYZ offsets so the G-code path starts at the current actual position
			IF poqDataIn <> 0 AND poqDataIn^.pbyBuffer <> 0 THEN
				fOffsetX := x_axis.fActPosition - poqDataIn^.pbyBuffer^[poqDataIn^.nReadPos].piStartPos.dX;
				fOffsetY := y_axis.fActPosition - poqDataIn^.pbyBuffer^[poqDataIn^.nReadPos].piStartPos.dY;
				fOffsetZ := z_axis.fActPosition - poqDataIn^.pbyBuffer^[poqDataIn^.nReadPos].piStartPos.dZ;
			END_IF
			iState := STATE_CNC_IPO;
		END_IF

	// Run the G-code interpolation on XYZ (offsets frozen on entry)
	STATE_CNC_IPO:
		poqDataIn := ADR(DEMO_GCODE);
		bExecute := TRUE;
		IF bDone OR bError THEN
			bExecute := FALSE;
			iState := STATE_IDLE;
		END_IF
END_CASE

END_PROGRAM

// xLH_base/app/IO/FB_XLH_GPIO
// =====================================================================
// FB_XLH_GPIO
// Pure data container for the GPIO control elements of the xLH board:
// 7 LEDs as inputs (written by the PLC program) and 8 switches as
// outputs (read from the board). The fields are mapped to the hardware
// via the device I/O configuration (CANopen); the read/write methods
// are currently empty and serve as extension hooks.
// =====================================================================
FUNCTION_BLOCK FB_XLH_GPIO
VAR_INPUT
	bLed1: BOOL;
	bLed2: BOOL;
	bLed3: BOOL;
	bLed4: BOOL;
	bLed5: BOOL;
	bLed6: BOOL;
	bLed7: BOOL;	
END_VAR
VAR_OUTPUT
	bSw1: BOOL;
	bSw2: BOOL;
	bSw3: BOOL;
	bSw4: BOOL;
	bSw5: BOOL;
	bSw6: BOOL;
	bSw7: BOOL;
	bSw8: BOOL;
END_VAR

METHOD read : BOOL
VAR_INPUT
END_VAR
END_METHOD

METHOD write : BOOL
VAR_INPUT
END_VAR
END_METHOD

END_FUNCTION_BLOCK

// xLH_base/app/IO/FB_XLH_TERMINAL
// =====================================================================
// FB_XLH_GPIO
// Pure data container for the GPIO control elements of the xLH board:
// 7 LEDs as inputs (written by the PLC program) and 8 switches as
// outputs (read from the board). The fields are mapped to the hardware
// via the device I/O configuration (CANopen); the read/write methods
// are currently empty and serve as extension hooks.
// =====================================================================
FUNCTION_BLOCK FB_XLH_TERMINAL
VAR_INPUT
	eRgbReset: RGB;
	eRgbManual: RGB;
	eRgbF1: RGB;
	eRgbF2: RGB;
	eRgbF3: RGB;
	
	eRgb1: RGB;
	eRgb2: RGB;
	eRgb3: RGB;
	eRgb4: RGB;
	eRgb5: RGB;
	eRgb6: RGB;
		
	eRgbAxXp: RGB;
	eRgbAxXm: RGB;
	eRgbAxYp: RGB;
	eRgbAxYm: RGB;
	eRgbAxZp: RGB;
	eRgbAxZm: RGB;
	eRgbAxCp: RGB;
	eRgbAxCm: RGB;
	
	eRgbMagnet: RGB;
	
	eRgbAxEncoderC: RGB;
	eRgbAxEncoderXY: RGB;
	eRgbAxEncoderZ: RGB;	
	
	eRgbVelMaster: RGB;	
	usBrightness: USINT := 100;
	
	{attribute 'displaymode':='hex'} 
	abyOutData1: ARRAY[0..7] OF BYTE;
	{attribute 'displaymode':='hex'}
	abyOutData2: ARRAY[0..7] OF BYTE;
	{attribute 'displaymode':='hex'}
	abyOutData3: ARRAY[0..7] OF BYTE;
	{attribute 'displaymode':='hex'}
	abyOutData4: ARRAY[0..7] OF BYTE;
END_VAR
VAR_OUTPUT
	bReset: BOOL;
	bManual: BOOL;
	bF1: BOOL;
	bF2: BOOL;
	bF3: BOOL;
	
	b1: BOOL;
	b2: BOOL;
	b3: BOOL;
	b4: BOOL;
	b5: BOOL;
	b6: BOOL;
	
	bAxXp: BOOL;
	bAxXm: BOOL;
	bAxYp: BOOL;
	bAxYm: BOOL;
	bAxZp: BOOL;
	bAxZm: BOOL;
	bAxCp: BOOL;
	bAxCm: BOOL;
	
	bMagnet: BOOL;
	bAxEncoderC: BOOL;
	bAxEncoderXY: BOOL;
	bAxEncoderZ: BOOL;

	bRtReset: BOOL;
	bRtManual: BOOL;
	bRtF1: BOOL;
	bRtF2: BOOL;
	bRtF3: BOOL;
	
	bRt1: BOOL;
	bRt2: BOOL;
	bRt3: BOOL;
	bRt4: BOOL;
	bRt5: BOOL;
	bRt6: BOOL;
	
	bRtAxXp: BOOL;
	bRtAxXm: BOOL;
	bRtAxYp: BOOL;
	bRtAxYm: BOOL;
	bRtAxZp: BOOL;
	bRtAxZm: BOOL;
	bRtAxCp: BOOL;
	bRtAxCm: BOOL;
	
	bRtMagnet: BOOL;
	bRtAxEnnoderC: BOOL;
	bRtAxEncoderXY: BOOL;
	bRtAxEncoderZ: BOOL;

	iAxEncoderC: INT;
	iAxEncoderXY: INT;
	iAxEncoderZ: INT;
	iVelMaster: INT;
	rVelMaster: LREAL;	

	{attribute 'displaymode':='hex'} 
	abyInData1: ARRAY[0..7] OF BYTE;
	{attribute 'displaymode':='hex'}
	abyInData2: ARRAY[0..7] OF BYTE;
	{attribute 'displaymode':='hex'}
	abyInData3: ARRAY[0..7] OF BYTE;
	{attribute 'displaymode':='hex'}
	abyInData4: ARRAY[0..7] OF BYTE;
END_VAR
VAR
	fbRtReset: R_TRIG;
	fbRtManual: R_TRIG;
	fbRtF1: R_TRIG;
	fbRtF2: R_TRIG;
	fbRtF3: R_TRIG;
	
	fbRt1: R_TRIG;
	fbRt2: R_TRIG;
	fbRt3: R_TRIG;
	fbRt4: R_TRIG;
	fbRt5: R_TRIG;
	fbRt6: R_TRIG;	
	
	fbRtAxXp: R_TRIG;
	fbRtAxXm: R_TRIG;
	fbRtAxYp: R_TRIG;
	fbRtAxYm: R_TRIG;
	fbRtAxZp: R_TRIG;
	fbRtAxZm: R_TRIG;
	fbRtAxCp: R_TRIG;
	fbRtAxCm: R_TRIG;
	
	fbRtMagnet: R_TRIG;
	fbRtAxEnnoderC: R_TRIG;
	fbRtAxEncoderXY: R_TRIG;
	fbRtAxEncoderZ: R_TRIG;
END_VAR

METHOD read : BOOL
VAR_INPUT
END_VAR
VAR
	unpackByte: MEM.UnpackByte;	
	value: UNION_BYTE_INT;
END_VAR
// PDO 1
unpackByte(byValue := abyInData1[0]);	
bReset := unpackByte.xBit0;
bAxEncoderC := unpackByte.xBit1;
bAxEncoderXY := unpackByte.xBit2;
bAxEncoderZ := unpackByte.xBit3;
bManual := unpackByte.xBit4;
b1 := unpackByte.xBit5;
b2 := unpackByte.xBit6;
b3 := unpackByte.xBit7;

unpackByte(byValue := abyInData1[1]);	
b4 := unpackByte.xBit0;
b5 := unpackByte.xBit1;
b6 := unpackByte.xBit2;

value.abyStream[0] := abyInData1[2];
value.abyStream[1] := abyInData1[3];
iAxEncoderC := value.iInt;

value.abyStream[0] := abyInData1[4];
value.abyStream[1] := abyInData1[5];
iAxEncoderXY := value.iInt;

value.abyStream[0] := abyInData1[6];
value.abyStream[1] := abyInData1[7];
iAxEncoderZ := value.iInt;


// PDO 2
unpackByte(byValue := abyInData2[0]);
bF1 := unpackByte.xBit0;
bAxCp := unpackByte.xBit1;
bAxYp := unpackByte.xBit2;
bAxZp := unpackByte.xBit3;
bF2 := unpackByte.xBit4;
bAxXm := unpackByte.xBit5;
bMagnet := unpackByte.xBit6;
bAxXp := unpackByte.xBit7;

unpackByte(byValue := abyInData2[1]);
bF3 := unpackByte.xBit0;
bAxCm := unpackByte.xBit1;
bAxYm := unpackByte.xBit2;	
bAxZm := unpackByte.xBit3;

value.abyStream[0] := abyInData2[2];
value.abyStream[1] := abyInData2[3];
iVelMaster := value.iInt;
rVelMaster := INT_TO_LREAL(iVelMaster) / 4095.0;

// Edge detection
fbRtReset(CLK:=bReset, Q=>bRtReset);
fbRtManual(CLK:=bManual, Q=>bRtManual);
fbRtF1(CLK:=bF1, Q=>bRtF1);
fbRtF2(CLK:=bF2, Q=>bRtF2);
fbRtF3(CLK:=bF3, Q=>bRtF3);
fbRt1(CLK:=b1, Q=>bRt1);
fbRt1(CLK:=b2, Q=>bRt2);
fbRt1(CLK:=b3, Q=>bRt3);
fbRt1(CLK:=b4, Q=>bRt4);
fbRt1(CLK:=b5, Q=>bRt5);
fbRt1(CLK:=b6, Q=>bRt6);
fbRtAxXp(CLK:=bAxXp, Q=>bRtAxXp);
fbRtAxXm(CLK:=bAxXm, Q=>bRtAxXm);
fbRtAxYp(CLK:=bAxYp, Q=>bRtAxYp);
fbRtAxYm(CLK:=bAxYm, Q=>bRtAxYm);
fbRtAxZp(CLK:=bAxZp, Q=>bRtAxZp);
fbRtAxZm(CLK:=bAxZm, Q=>bRtAxZm);
fbRtAxCp(CLK:=bAxCp, Q=>bRtAxCp);
fbRtAxCm(CLK:=bAxCm, Q=>bRtAxCm);
fbRtMagnet(CLK:=bMagnet, Q=>bRtMagnet);
fbRtAxEnnoderC(CLK:=bAxEncoderC, Q=>bRtAxEnnoderC);
fbRtAxEncoderXY(CLK:=bAxEncoderXY, Q=>bRtAxEncoderXY);
fbRtAxEncoderZ(CLK:=bAxEncoderZ, Q=>bRtAxEncoderZ);
END_METHOD

METHOD write : BOOL
VAR_INPUT
END_VAR
abyOutData1[0] := MEM.PackBitsToByte(
	((eRgbAxEncoderZ = RGB.GREEN) OR (eRgbAxEncoderZ = RGB.BLUE)),
	((eRgbAxEncoderZ = RGB.RED) OR (eRgbAxEncoderZ = RGB.BLUE)),
	//
	((eRgbAxEncoderXY = RGB.GREEN) OR (eRgbAxEncoderXY = RGB.BLUE)),
	((eRgbAxEncoderXY = RGB.RED) OR (eRgbAxEncoderXY = RGB.BLUE)),
	//
	((eRgbAxEncoderC = RGB.GREEN) OR (eRgbAxEncoderC = RGB.BLUE)),
	((eRgbAxEncoderC = RGB.RED) OR (eRgbAxEncoderC = RGB.BLUE)),
	//
	((eRgbReset = RGB.GREEN) OR (eRgbReset = RGB.BLUE)),
	((eRgbReset = RGB.RED) OR (eRgbReset = RGB.BLUE)));


abyOutData1[1] := MEM.PackBitsToByte(
	((eRgb3 = RGB.GREEN) OR (eRgb3 = RGB.BLUE)),
	((eRgb3 = RGB.RED) OR (eRgb3 = RGB.BLUE)),
	//
	((eRgb2 = RGB.GREEN) OR (eRgb2 = RGB.BLUE)),
	((eRgb2 = RGB.RED) OR (eRgb2 = RGB.BLUE)),
	//
	((eRgb1 = RGB.GREEN) OR (eRgb1 = RGB.BLUE)),
	((eRgb1 = RGB.RED) OR (eRgb1 = RGB.BLUE)),
	//
	((eRgbManual = RGB.GREEN) OR (eRgbManual = RGB.BLUE)),
	((eRgbManual = RGB.RED) OR (eRgbManual = RGB.BLUE)));


abyOutData1[2] := MEM.PackBitsToByte(
	((eRgbF1 = RGB.GREEN) OR (eRgbF1 = RGB.BLUE)),
	((eRgbF1 = RGB.RED) OR (eRgbF1 = RGB.BLUE)),
	//
	((eRgb6 = RGB.GREEN) OR (eRgb6 = RGB.BLUE)),
	((eRgb6 = RGB.RED) OR (eRgb6 = RGB.BLUE)),
	//
	((eRgb5 = RGB.GREEN) OR (eRgb5 = RGB.BLUE)),
	((eRgb5 = RGB.RED) OR (eRgb5 = RGB.BLUE)),
	//
	((eRgb4 = RGB.GREEN) OR (eRgb4 = RGB.BLUE)),
	((eRgb4 = RGB.RED) OR (eRgb4 = RGB.BLUE)));	
	


abyOutData1[3] := MEM.PackBitsToByte(
	((eRgbF2 = RGB.GREEN) OR (eRgbF2 = RGB.BLUE)),
	((eRgbF2 = RGB.RED) OR (eRgbF2 = RGB.BLUE)),
	//
	((eRgbAxZp = RGB.GREEN) OR (eRgbAxZp = RGB.BLUE)),
	((eRgbAxZp = RGB.RED) OR (eRgbAxZp = RGB.BLUE)),
	//
	((eRgbAxYp = RGB.GREEN) OR (eRgbAxYp = RGB.BLUE)),
	((eRgbAxYp = RGB.RED) OR (eRgbAxYp = RGB.BLUE)),
	//
	((eRgbAxCp = RGB.GREEN) OR (eRgbAxCp = RGB.BLUE)),
	((eRgbAxCp = RGB.RED) OR (eRgbAxCp = RGB.BLUE)));	



abyOutData1[4] := MEM.PackBitsToByte(
	((eRgbAxXp = RGB.GREEN) OR (eRgbAxXp = RGB.BLUE)),
	((eRgbAxXp = RGB.RED) OR (eRgbAxXp = RGB.BLUE)),
	//
	((eRgbMagnet = RGB.GREEN) OR (eRgbMagnet = RGB.BLUE)),
	((eRgbMagnet = RGB.RED) OR (eRgbMagnet = RGB.BLUE)),
	//
	((eRgbAxXm = RGB.GREEN) OR (eRgbAxXm = RGB.BLUE)),
	((eRgbAxXm = RGB.RED) OR (eRgbAxXm = RGB.BLUE)),
	//
	((eRgbVelMaster = RGB.GREEN) OR (eRgbVelMaster = RGB.BLUE)),
	((eRgbVelMaster = RGB.RED) OR (eRgbVelMaster = RGB.BLUE)));
	
	
abyOutData1[5] := MEM.PackBitsToByte(
	((eRgbAxZm = RGB.GREEN) OR (eRgbAxZm = RGB.BLUE)),
	((eRgbAxZm = RGB.RED) OR (eRgbAxZm = RGB.BLUE)),
	//
	((eRgbAxYm = RGB.GREEN) OR (eRgbAxYm = RGB.BLUE)),
	((eRgbAxYm = RGB.RED) OR (eRgbAxYm = RGB.BLUE)),
	//
	((eRgbAxCm = RGB.GREEN) OR (eRgbAxCm = RGB.BLUE)),
	((eRgbAxCm = RGB.RED) OR (eRgbAxCm = RGB.BLUE)),
	//
	((eRgbF3 = RGB.GREEN) OR (eRgbF3 = RGB.BLUE)),
	((eRgbF3 = RGB.RED) OR (eRgbF3 = RGB.BLUE)));
	
abyOutData1[7] := usBrightness;
END_METHOD

END_FUNCTION_BLOCK

// xLH_base/app/IO/FB_XLH_MOTION
// =====================================================================
// FB_XLH_MOTION
// Aggregate container for all motion I/Os of the xLH board (4 stepper
// axes, limit switches/sensor, 8 servo channels, magnet PWM, frequency
// outputs). Mapped to the motion hardware via CANopen PDOs.
//
// mRead()  calls per axis fbAxisPlcOpen() (PLCopen FB), the axis FB
// itself, passes the encoder position (adiPosition) and calls mRead.
// mWrite() calls per axis mWrite, packs _bDir/_bEn/_bInMotion etc. into
// abyControl[i], computes the pulse frequency from _diFrequency in the
// range [fFREQ_OUT_MIN, fFREQ_OUT_MAX] and smooths the value with a
// per-axis Kalman filter before writing it to adiFrequency[i].
//
// Stepper motor:
//   Pulses per revolution = 64 * 400 = 25600
// Drive x y z:
//   Diameter 10.0012925 mm
//   Pulses per mm = 25600 / (d * pi) = 814.768
// Conveyor:
//   Gear ratio 3/1
//   Pulses per mm = 3 * 25600 / (d * pi) = 660.708
// =====================================================================
FUNCTION_BLOCK FB_XLH_MOTION
VAR_INPUT
	adiPosition: ARRAY[1..4] OF DINT;
	{attribute 'displaymode':='bin'} 
	abyInputs: ARRAY[1..3] OF BYTE;
	bAxXsw: BOOL;
	bAxYsw: BOOL;
	bAxZsw: BOOL;
	bSensor: BOOL;
	_bSensorHw: BOOL;
	bSensorConveyorFront: BOOL;
	_bSensorConveyorFrontHw: BOOL;
	bSensorConveyorBack: BOOL;
	_bSensorConveyorBackHw: BOOL;
	
	
	{attribute 'displaymode':='bin'} 
	abyControl: ARRAY[1..4] OF BYTE;
	afFrequencyCalc: ARRAY[1..4] OF LREAL;
	afbFilterFrequency: ARRAY[1..4] OF FB_KALMAN_FILTER;
	adiFrequency: ARRAY[1..4] OF DINT;
	uiMagnetDutyCycle: UINT;
	abyOutputs: ARRAY[1..2] OF BYTE;
	ausServo: ARRAY[1..8] OF USINT;
	
	pfbXlhMotionAxis: ARRAY [1..4] OF POINTER TO FB_XLH_MOTION_AXIS_BASE;
END_VAR
VAR_OUTPUT
END_VAR
VAR CONSTANT
	fCLK_HZ          : LREAL := 150000000.0;
	fSTEP_PERIOD_MIN : REAL := 0.25;
	fSTEP_PERIOD_MAX : REAL := 50000.0;
	fFREQ_OUT_MIN    : LREAL := 2000.0;
	fFREQ_OUT_MAX    : LREAL := 600000000.0;
END_VAR

METHOD read : BOOL
VAR
	i: INT;
END_VAR
FOR i := 1 TO 4 DO
	pfbXlhMotionAxis[i]^.fbAxisPlcOpen();
	pfbXlhMotionAxis[i]^();
	pfbXlhMotionAxis[i]^.diPosition := adiPosition[i];
	pfbXlhMotionAxis[i]^.mRead();
END_FOR

bSensor := NOT _bSensorHw;
bSensorConveyorFront := NOT _bSensorConveyorFrontHw;
bSensorConveyorBack := NOT _bSensorConveyorBackHw;
END_METHOD

METHOD write : BOOL
VAR
	i: INT;
END_VAR
FOR i := 1 TO 4 DO
	pfbXlhMotionAxis[i]^.mWrite();

	abyControl[i] := MEM.PackBitsToByte(
		FALSE,
		FALSE,
		pfbXlhMotionAxis[i]^.bMoveWithoutPulse,
		pfbXlhMotionAxis[i]^._bInMotion,
		pfbXlhMotionAxis[i]^.bInverted,
		pfbXlhMotionAxis[i]^.bReset,
		pfbXlhMotionAxis[i]^._bDir,
		pfbXlhMotionAxis[i]^._bEn);

	afFrequencyCalc[i] := fCLK_HZ / LIMIT(fSTEP_PERIOD_MIN, TO_REAL(pfbXlhMotionAxis[i]^._diFrequency), fSTEP_PERIOD_MAX);
	afbFilterFrequency[i](fX:=afFrequencyCalc[i], fR:=1.0, fQ:=1.0);
	adiFrequency[i] := LREAL_TO_DINT(LIMIT(fFREQ_OUT_MIN, afbFilterFrequency[i].fY, fFREQ_OUT_MAX));
END_FOR
END_METHOD

END_FUNCTION_BLOCK

// xLH_base/app/MOTION_BASE/FB_KALMAN_FILTER
// =====================================================================
// FB_KALMAN_FILTER
// One-dimensional discrete Kalman filter for smoothing scalar
// measurement signals. Inputs: fX (measurement), fQ (process noise),
// fR (measurement noise), bReset to clear the internal states.
// Output fY is the estimated quantity X_hat. The bias fAvoidZero
// prevents a division by zero when computing K.
// Used e.g. in FB_XLH_MOTION to smooth the pulse-frequency
// calculation.
// =====================================================================
FUNCTION_BLOCK PUBLIC FB_KALMAN_FILTER
VAR_INPUT
	fX: LREAL;
	fQ: LREAL;
	fR: LREAL;
	bReset: BOOL;
END_VAR
VAR_OUTPUT
	fY: LREAL;
END_VAR
VAR 
	X_hat: LREAL;
	X_hat_min: LREAL;
	poise: LREAL;
	Pmin: LREAL;
	K: LREAL;
END_VAR
VAR CONSTANT
	fAvoidZero: LREAL := 0.001;
END_VAR

IF bReset THEN
	reset();
END_IF

K := Pmin/MAX((Pmin + fR), fAvoidZero);
X_hat := X_hat_min + K*(fX - X_hat_min);
poise := (1 - K)*Pmin;
Pmin := poise + fQ;
X_hat_min := X_hat;
fY := X_hat;

ACTION reset:
X_hat := 0.0;
X_hat_min := 0.0;
poise := 0.0;
Pmin := 0.0;
K := 0.0;
fY := 0.0;
END_ACTION

END_FUNCTION_BLOCK

// xLH_base/app/MOTION_BASE/FB_XLH_MOTION_AXIS_BASE
// =====================================================================
// FB_XLH_MOTION_AXIS_BASE
// Base class for the hardware interface between a stepper-motor axis
// and the SoftMotion layer. Method mRead() writes the raw encoder
// position (diPosition) into the AXIS_REF_POSCONTROL and reports
// drive/regulator status. mWrite() computes from the SoftMotion-provided
// target velocity (out.diSetVelocity) the pulse frequency, the
// direction bit (_bDir), the enable (_bEn) and the filtered
// in-motion flag (_bInMotion). Extended by FB_XLH_MOTION_AXIS_SIMPLE
// and FB_XLH_MOTION_AXIS_SIMPLE_ES.
// =====================================================================
FUNCTION_BLOCK FB_XLH_MOTION_AXIS_BASE
VAR_INPUT
	bInverted: BOOL;
	bReset: BOOL;
	bMoveWithoutPulse: BOOL;
	diPosition: DINT;
	pAxis: POINTER TO AXIS_REF_POSCONTROL;
	fbAxisPlcOpen: REFERENCE TO FB_PLC_OPEN_AXIS;
END_VAR
VAR_OUTPUT
	
END_VAR
VAR
	_fbTofSm1: TOF;
	_bEn: BOOL;
	_bDir: BOOL;
	_bInMotion: BOOL;
	_diFrequency: DINT;
END_VAR

METHOD mRead : BOOL
IF pAxis > 16#0 THEN
	pAxis^.in.dwActPosition := TO_DWORD(diPosition);
	pAxis^.in.bDriveStartRealState := TRUE;
	pAxis^.in.bRegulatorRealState := TRUE;
END_IF
END_METHOD

METHOD mWrite : BOOL
IF pAxis > 16#0 THEN
	_bDir := (pAxis^.out.diSetVelocity >= 0);
	_diFrequency := ABS(pAxis^.out.diSetVelocity);
	// https://content.helpme-codesys.com/en/libs/SM3_Basic/Current/SM3_Basic/DataTypes/DriveInterface/SMC_AXIS_STATE.html
	_bEn := (pAxis^.nAxisState >= 1);
	_fbTofSm1(IN:=(pAxis^.nAxisState >= 4), PT:=T#1000MS, Q=>_bInMotion);
END_IF
END_METHOD

END_FUNCTION_BLOCK

// xLH_base/app/MOTION_BASE/FB_XLH_MOTION_AXIS_SIMPLE
// =====================================================================
// FB_XLH_MOTION_AXIS_SIMPLE
// Simple homing without a limit switch: moves the axis at
// fVelHoming*10 absolutely to position 0 (with bMoveWithoutPulse, i.e.
// only the setpoint is updated, no pulses are emitted), waits for a
// settling period and reports bHomingDone. Used for the A axis, which
// has no physical limit switch.
// Extends FB_XLH_MOTION_AXIS_BASE.
// =====================================================================
FUNCTION_BLOCK FB_XLH_MOTION_AXIS_SIMPLE EXTENDS FB_XLH_MOTION_AXIS_BASE
VAR_INPUT
	bHoming: BOOL;
	fVelHoming: LREAL;
	eMcHomingDirection: MC_Direction;
END_VAR
VAR_OUTPUT
	bHomingDone: BOOL;
END_VAR
VAR
	iState: INT;
	fbTonDelay1: TON;
END_VAR
VAR CONSTANT
	iSTATE_IDLE      : INT := 0;
	iSTATE_GOTO_ZERO : INT := 100;
	iSTATE_SETTLE    : INT := 110;
	iSTATE_DONE      : INT := 120;
END_VAR

SUPER^();
bReset := FALSE;
bMoveWithoutPulse := FALSE;
bHomingDone := FALSE;

IF NOT bHoming THEN
	iState := iSTATE_IDLE;
END_IF

IF __ISVALIDREF(fbAxisPlcOpen) THEN
	CASE iState OF
		iSTATE_IDLE:
			IF bHoming THEN
				iState := iSTATE_GOTO_ZERO;
			END_IF

		iSTATE_GOTO_ZERO:
			bReset := TRUE;
			bMoveWithoutPulse := TRUE;
			fbAxisPlcOpen.fVel := fVelHoming * 10.0;
			fbAxisPlcOpen.mcma.Execute := TRUE;
			fbAxisPlcOpen.mcma.Position := 0.0;
			IF fbAxisPlcOpen.mcma.Done THEN
				fbAxisPlcOpen.executeToFalse();
				iState := iSTATE_SETTLE;
			END_IF

		iSTATE_SETTLE:
			bReset := TRUE;
			bMoveWithoutPulse := TRUE;
			IF fbTonDelay1.Q THEN
				iState := iSTATE_DONE;
			END_IF

		iSTATE_DONE:
			bHomingDone := TRUE;

	ELSE
		iState := iSTATE_IDLE;
	END_CASE
ELSE
	iState := iSTATE_IDLE;
END_IF

fbTonDelay1(IN := iState = iSTATE_SETTLE, PT := T#100MS);

END_FUNCTION_BLOCK

// xLH_base/app/MOTION_BASE/FB_XLH_MOTION_AXIS_SIMPLE_ES
// =====================================================================
// FB_XLH_MOTION_AXIS_SIMPLE_ES
// Homing with a limit switch (state machine):
//   FAST_SEEK   -> fast search at fVelHomingFast until the limit switch
//   FAST_STOP   -> stop, then
//   RETREAT     -> short retreat by rOFFSET_HOMING
//   SLOW_SEEK   -> slow search at fVelHoming until the limit switch
//   SLOW_STOP   -> stop, then
//   MOVE_OFFSET -> traverse by fOffset (machine zero correction)
//   GOTO_ZERO   -> set the setpoint position to 0 (no pulses emitted)
//   SETTLE      -> 250 ms settle
//   DONE        -> bHomingDone := TRUE
// Used for the X/Y/Z axes with limit switch (pbEs points to the
// respective limit-switch signal). Extends FB_XLH_MOTION_AXIS_BASE.
// =====================================================================
FUNCTION_BLOCK FB_XLH_MOTION_AXIS_SIMPLE_ES EXTENDS FB_XLH_MOTION_AXIS_BASE
VAR_INPUT
	bHoming: BOOL;
	fVelHoming: LREAL;
	fVelHomingFast: LREAL;
	eMcHomingDirection: MC_Direction;
	fOffset: LREAL;
	fPosition: LREAL;
	pbEs: POINTER TO BOOL;
END_VAR
VAR_OUTPUT
	bHomingDone: BOOL;
	bEs: BOOL;
END_VAR
VAR
	iState: INT;
	fbTonDelay1: TON;
END_VAR
VAR CONSTANT
	rOFFSET_HOMING: REAL := 3.0;

	iSTATE_IDLE        : INT := 0;
	iSTATE_FAST_SEEK   : INT := 100;
	iSTATE_FAST_STOP   : INT := 110;
	iSTATE_RETREAT     : INT := 120;
	iSTATE_SLOW_SEEK   : INT := 130;
	iSTATE_SLOW_STOP   : INT := 140;
	iSTATE_MOVE_OFFSET : INT := 150;
	iSTATE_GOTO_ZERO    : INT := 160;
	iSTATE_SETTLE      : INT := 170;
	iSTATE_DONE        : INT := 180;
END_VAR

SUPER^();
bReset := FALSE;
bMoveWithoutPulse := FALSE;
bHomingDone := FALSE;

IF NOT bHoming THEN
	iState := iSTATE_IDLE;
END_IF

IF __ISVALIDREF(fbAxisPlcOpen) THEN
	CASE iState OF
		iSTATE_IDLE:
			IF bHoming THEN
				iState := iSTATE_FAST_SEEK;
			END_IF

		iSTATE_FAST_SEEK:
			fbAxisPlcOpen.fVel := fVelHomingFast;
			fbAxisPlcOpen.mcmv.Execute := TRUE;
			fbAxisPlcOpen.mcmv.Direction := eMcHomingDirection;
			IF NOT bEs THEN
				fbAxisPlcOpen.executeToFalse();
				iState := iSTATE_FAST_STOP;
			END_IF

		iSTATE_FAST_STOP:
			fbAxisPlcOpen.mcs.Execute := TRUE;
			IF fbAxisPlcOpen.mcs.Done THEN
				fbAxisPlcOpen.executeToFalse();
				iState := iSTATE_RETREAT;
			END_IF

		iSTATE_RETREAT:
			fbAxisPlcOpen.fVel := fVelHoming;
			fbAxisPlcOpen.mcmr.Execute := TRUE;
			IF eMcHomingDirection = MC_Direction.negative THEN
				fbAxisPlcOpen.mcmr.Distance := rOFFSET_HOMING;
			ELSE
				fbAxisPlcOpen.mcmr.Distance := -rOFFSET_HOMING;
			END_IF
			IF fbAxisPlcOpen.mcmr.Done THEN
				fbAxisPlcOpen.executeToFalse();
				iState := iSTATE_SLOW_SEEK;
			END_IF

		iSTATE_SLOW_SEEK:
			fbAxisPlcOpen.fVel := fVelHoming;
			fbAxisPlcOpen.mcmv.Execute := TRUE;
			fbAxisPlcOpen.mcmv.Direction := eMcHomingDirection;
			IF NOT bEs THEN
				fbAxisPlcOpen.executeToFalse();
				iState := iSTATE_SLOW_STOP;
			END_IF

		iSTATE_SLOW_STOP:
			fbAxisPlcOpen.mcs.Execute := TRUE;
			IF fbAxisPlcOpen.mcs.Done THEN
				fbAxisPlcOpen.executeToFalse();
				iState := iSTATE_MOVE_OFFSET;
			END_IF

		iSTATE_MOVE_OFFSET:
			fbAxisPlcOpen.fVel := TO_REAL(fbAxisPlcOpen.pAxis^.fSWMaxVelocity);
			fbAxisPlcOpen.mcmr.Execute := TRUE;
			fbAxisPlcOpen.mcmr.Distance := fOffset;
			IF fbAxisPlcOpen.mcmr.Done THEN
				fbAxisPlcOpen.executeToFalse();
				iState := iSTATE_GOTO_ZERO;
			END_IF

		iSTATE_GOTO_ZERO:
			bMoveWithoutPulse := TRUE;
			fbAxisPlcOpen.fVel := TO_REAL(fbAxisPlcOpen.pAxis^.fSWMaxVelocity);
			fbAxisPlcOpen.mcma.Execute := TRUE;
			fbAxisPlcOpen.mcma.Position := 0.0;
			IF fbAxisPlcOpen.mcma.Done THEN
				fbAxisPlcOpen.executeToFalse();
				iState := iSTATE_SETTLE;
			END_IF

		iSTATE_SETTLE:
			bMoveWithoutPulse := TRUE;
			IF fbTonDelay1.Q THEN
				iState := iSTATE_DONE;
			END_IF

		iSTATE_DONE:
			bHomingDone := TRUE;

	ELSE
		iState := iSTATE_IDLE;
	END_CASE
ELSE
	iState := iSTATE_IDLE;
END_IF

fbTonDelay1(IN := iState = iSTATE_SETTLE, PT := T#500MS);

METHOD mRead : BOOL
SUPER^.mRead();
IF pbEs > 16#0 THEN
	bEs := pbEs^;
ELSE
	bEs := FALSE;
END_IF
END_METHOD

END_FUNCTION_BLOCK

// xLH_base/app/MAIN_CALLER
PROGRAM MAIN_CALLER
VAR
	bDevicesCoRunning: BOOL;
	fbTonDevicesCoRunning: TON := (PT:=T#250MS);
	
END_VAR

// Monitor whether all CANopen devices are in the RUN state

fbTonDevicesCoRunning(IN:= 
	(xlh_motion.CANopenState = _3SCOS.DEVICE_STATE.OPERATIONAL) AND
	(xlh_terminal.CANopenState = _3SCOS.DEVICE_STATE.OPERATIONAL)	
);

(*
fbTonDevicesCoRunning(IN:= 
	(xlh_motion.CANopenState = _3SCOS.DEVICE_STATE.OPERATIONAL)
);
*)
IF fbTonDevicesCoRunning.Q THEN
	bDevicesCoRunning := TRUE;
END_IF

// if all devices are in the RUN state (including the debounce delay), the MAIN POU is called
IF bDevicesCoRunning THEN
	MC();
END_IF

END_PROGRAM

// xLH_base/app/Visualization
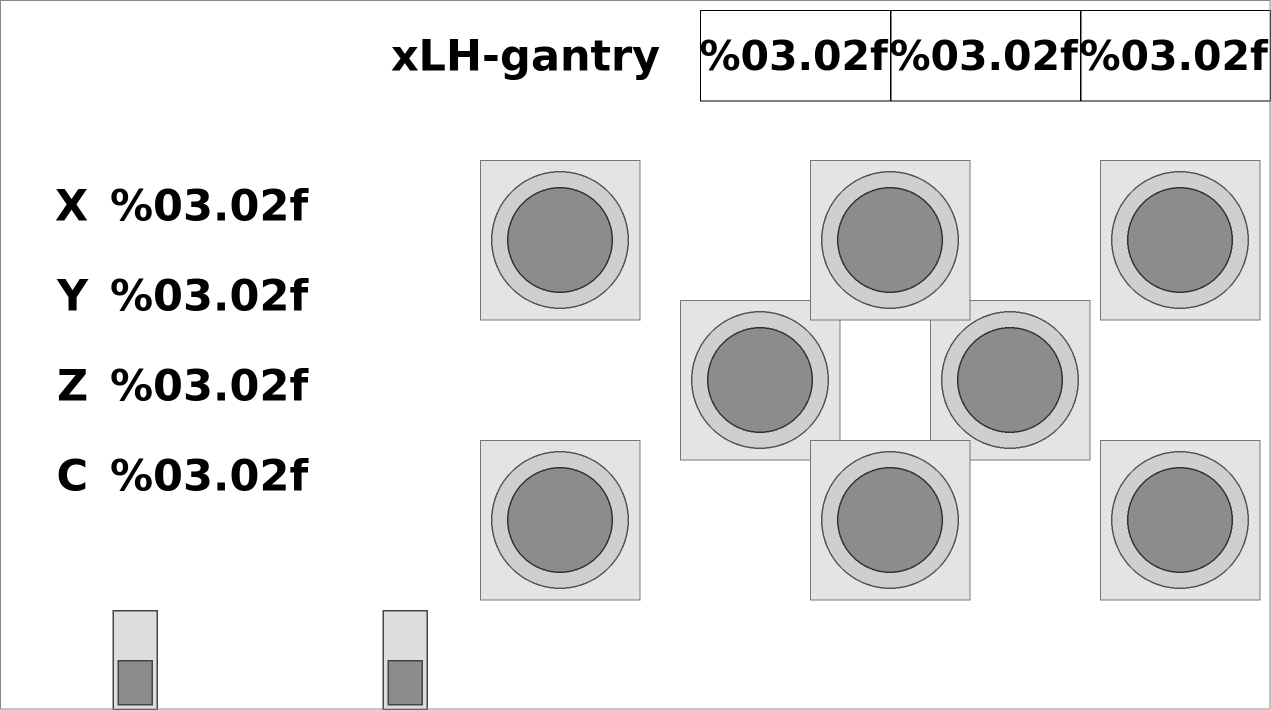
VISUALIZATION Visualization  // 1271x710
    PushSwitch (680,300 160x160), variable: MANUAL_MODE.bXm, behaviour: TAP, style: Switch-PushSwitch-Gray
    PushSwitch (930,300 160x160), variable: MANUAL_MODE.bXp, behaviour: TAP, style: Switch-PushSwitch-Gray
    PushSwitch (810,160 160x160), variable: MANUAL_MODE.bYp, behaviour: TAP, style: Switch-PushSwitch-Gray
    PushSwitch (810,440 160x160), variable: MANUAL_MODE.bYm, behaviour: TAP, style: Switch-PushSwitch-Gray
    PushSwitch (1100,160 160x160), variable: MANUAL_MODE.bZp, behaviour: TAP, style: Switch-PushSwitch-Gray
    PushSwitch (1100,440 160x160), variable: MANUAL_MODE.bZm, behaviour: TAP, style: Switch-PushSwitch-Gray
    Rectangle (90,160 221x91), "%03.02f", text variable: MC.axX.fActPos
    Rectangle (0,10 1051x91), "xLH-gantry"
    Rectangle (10,160 81x91), "X"
    Rectangle (90,250 221x91), "%03.02f", text variable: MC.axY.fActPos
    Rectangle (10,250 81x91), "Y"
    Rectangle (90,340 221x91), "%03.02f", text variable: MC.axZ.fActPos
    Rectangle (10,340 81x91), "Z"
    Rectangle (1080,10 191x91), "%03.02f", text variable: MANUAL_MODE.fStepZ
        OnMouseClick: write the text variable via VisuDialogs.Numpad, min 0.1, max 50.0
    DipSwitch (10,610 250x100), variable: io.bMagnet, behaviour: TOGGLE, style: Switch-DipSwitch-Gray
    DipSwitch (280,610 250x100), variable: APP_SQUARE_MODE.bStart, behaviour: TOGGLE, style: Switch-DipSwitch-Gray
    PushSwitch (480,160 160x160), variable: MANUAL_MODE.bCp, behaviour: TAP, style: Switch-PushSwitch-Gray
    PushSwitch (480,440 160x160), variable: MANUAL_MODE.bCm, behaviour: TAP, style: Switch-PushSwitch-Gray
    Rectangle (90,430 221x91), "%03.02f", text variable: MC.axC.fActPos
    Rectangle (10,430 81x91), "C"
    Rectangle (890,10 191x91), "%03.02f", text variable: MANUAL_MODE.fStepXY
        OnMouseClick: write the text variable via VisuDialogs.Numpad, min 0.1, max 50.0
    Rectangle (700,10 191x91), "%03.02f", text variable: MANUAL_MODE.fStepC
        OnMouseClick: write the text variable via VisuDialogs.Numpad, min 0.1, max 50.0
END_VISUALIZATION

(* text DEMO_GCODE
N000 G01 X0 Y0 Z0 E100 E-100 F15
N010 G00 X-25 Y0 
N020 G01 Z-5.0 
N030 G01 X-25 Y22.5 
N040 G02 X-22.5 Y25 I2.5 J0 
N050 G01 X-15 Y25 
N060 G02 X15 Y25 I15 J0 K180 
N070 G01 X22.5 Y25 
N080 G02 X25 Y22.5 I0 J-2.5 
N090 G01 X25 Y0 
N100 G01 X-25 Y0 
N110 G00 Z10 
N120 G00 X-11.25 Y12.5 
N130 G00 Z-10.0 
N140 G02 I-5 J0 
N150 G00 Z10 
N160 G00 X11.25 Y12.5 
N170 G00 Z-10.0 
N180 G02 I5 J0
N190 G00 Z10 
N200 G00 X0 Y0
*)
